	// Only enabled zones are considered
	ELSIF ZoneTable[mIdx].Used THEN
		// Only empty zones are considered and not marked to be flushed
		IF NOT ZoneTable[mIdx].TU_Present AND NOT ZoneTable[mIdx].Flush THEN
			// A zone candidate needs to provide the right length and is not reserver already
			IF ZoneTable[mIdx].ActionId = 0 AND
               ZoneTable[mIdx].ZoneLength >=  mLength THEN
				// When start position of zone is higher, the position is in front of the requested position
				// All others are after overflow point
				IF ZoneTable[mIdx].ZoneStartPosition >= mTrackingPosition THEN
					mDistanceToCurrentZone := ZoneTable[mIdx].ZoneStartPosition - mTrackingPosition;
					
					// Check if distance in a valid range for assignment
					IF mDistanceToCurrentZone <= mMaxAssignDistance THEN
						IF mDistanceToLastFoundZone > mDistanceToCurrentZone THEN
							mDistanceToLastFoundZone := mDistanceToCurrentZone;
							mFoundZoneIndex := mIdx;
						END_IF
					END_IF
				ELSE
					mDistanceToCurrentZone := ZoneTable[mIdx].ZoneStartPosition + TotalTrackingLength - mTrackingPosition;
				
					// Check if distance in a valid range for assignment
					IF mDistanceToCurrentZone <= mMaxAssignDistance THEN
						IF mDistanceToLastFoundZone > mDistanceToCurrentZone THEN
							mDistanceToLastFoundZone := mDistanceToCurrentZone;
							mFoundZoneIndex := mIdx;
						END_IF
					END_IF
				END_IF
			END_IF
		END_IF
		
		mZoneCounter := mZoneCounter + 1;
	END_IF	
END_FOR

// Reserve zone
IF mFoundZoneIndex > 0 THEN
	ZoneTable[mFoundZoneIndex].ActionId := mActionId;
	ZoneTable[mFoundZoneIndex].iActionListener := miActionListener;
	ZoneTable[mFoundZoneIndex].PositionToLive := mPositionToLive;
	
	// When a position to live is configured, ensure zone gets monitored
	IF mPositionToLive > 0 THEN
		M_AddZoneToPTL(mFoundZoneIndex);
	ELSE
		// It is possible that found zone had already a PTL
		// If new one is 0, means no monitoring
		M_RemoveZoneFromPTL(mFoundZoneIndex);
	END_IF
END_IF

M_AssignNextFreeZone := mFoundZoneIndex;
END_METHOD

/// Calculates full tracking distance and ensure its a multiple of windowsize.
/// Additional it adds the tracking addition distance to allow more space for reservations.
METHOD PROTECTED M_CalculateTotalTrackingLength : UDINT // Returns complete tracking distance 
VAR_INPUT
	mTrackingLength			: UDINT; // Length of tracking segment [mm] (e.g. conveyor length)
	mTrackingAddition		: UDINT; // Additional tracking length [mm]
	mWindowSize				: UINT; // Window size [mm]
END_VAR
VAR
	mLength					: UDINT; // Tracking length with out taking care of window size
	mRest					: UDINT; // Missing value between Length and next integer
END_VAR
(* Calculation is based on the following:
	+ 2 * Tracking length
	+ Tracking addition
	+ supplement to ensure its a multiple of window size
*)

mLength := mTrackingLength * 2 + TrackingAddition;
mRest := mLength MOD mWindowSize;

IF mRest > 0 THEN
	M_CalculateTotalTrackingLength := mLength + (mWindowSize-mRest);
ELSE
	M_CalculateTotalTrackingLength := mLength;
END_IF
END_METHOD

/// Clears all windows, zones and ongoing transfers. Notifies all listeners.
/// Remark: This method is executed immediately and can therefore influence
///         ongoing operations.
METHOD M_ClearTables : BOOL // Returns true if successful, otherwise false
VAR
	mZoneCounter		: INT;
	mIdx				: UINT;
END_VAR
VAR_INST
	AllTablesCleared	: BOOL;
	OldZoneTable		: ARRAY[1..MAX_NUMBER_OF_ZONES] OF ST_WindowTrackingZone; // List of all zones
END_VAR
M_ClearTables := FALSE;

// Store old zone table
OldZoneTable := ZoneTable;

// Clear all tables
AllTablesCleared := MEMSET(ADR(WindowTable), 0, SIZEOF(WindowTable)) > 0 AND
				    MEMSET(ADR(ZoneTable), 0, SIZEOF(ZoneTable)) > 0 AND
				    MEMSET(ADR(OngoingTransferList), 0, SIZEOF(OngoingTransferList)) > 0 AND
				    MEMSET(ADR(PTL_Zones), 0, SIZEOF(PTL_Zones)) > 0;

// Inform listener
IF AllTablesCleared THEN
	mZoneCounter := 0;
	// Notify listeners
	FOR mIdx := 1 TO MAX_NUMBER_OF_ZONES DO
		// When number of present zone is reached
		IF mZoneCounter >= ZoneCount THEN
			EXIT;
			
		ELSIF OldZoneTable[mIdx].Used THEN
			// Check if zone had a registred action lister and notify
			IF OldZoneTable[mIdx].iActionListener <> 0 THEN
				OldZoneTable[mIdx].iActionListener.M_ActionZoneDeletedEvent(mIdx,OldZoneTable[mIdx]);
			END_IF
			
			// Inform window tracking listener
			IF iEventListener <> 0 THEN
				IF OldZoneTable[mIdx].TU_Present THEN
					iEventListener.M_TrackingTU_DeletedEvent(mIdx,OldZoneTable[mIdx]);
				END_IF
				
				iEventListener.M_TrackingZoneDeletedEvent(mIdx,OldZoneTable[mIdx]);
			END_IF
	
			mZoneCounter := mZoneCounter + 1;	
		END_IF
	END_FOR
	
	// Clean internal counters
	ZoneCount := 0;
	TU_Count := 0;
	
	M_ClearTables := TRUE;
END_IF
END_METHOD

/// Clears window and initialize with default values
METHOD PROTECTED M_ClearWindow : BOOL // returns true if successfull cleared, otherwise false
VAR_INPUT
	mWindowIndex	: UINT; // Window index to clear
END_VAR
M_ClearWindow := FALSE;

// Validate inputs
IF mWindowIndex <= 0 OR
   mWindowIndex > MaxWindowIndex THEN
   RETURN;
END_IF

M_ClearWindow := MEMSET(ADR(WindowTable[mWindowIndex]), 0, SIZEOF(WindowTable[mWindowIndex])) > 0;
END_METHOD

/// Delete a zone and all related windows
/// Remark: Including zones with physical TUs 
METHOD M_DeleteZone : BOOL // Returns true if successful, otherwise false
VAR_INPUT
	mZoneIndex 				: UINT; // Zone index to delete
END_VAR
VAR
	mIdx					: UINT; // Loop iterator
	mZoneWindowLength 		: UINT; // Length of zone to be moved
	mWindowIndex			: UINT; // Start window index
	mDeletedOnTransferList	: BOOL; // Zone was found and deleted on transfer list
	mDeletedOnPTL			: BOOL; // Zone was found and deleted in PTL list
END_VAR
VAR_INST
	OldZoneData				: ST_WindowTrackingZone; // Old deleted zone data
END_VAR
M_DeleteZone := FALSE;

// Validate inputs
IF mZoneIndex <= 0 OR
   mZoneIndex > MAX_NUMBER_OF_ZONES THEN
   RETURN;
END_IF

// Check if zone is complete
IF ZoneTable[mZoneIndex].ZoneEndWindowIndex > 0 AND
   ZoneTable[mZoneIndex].ZoneStartWindowIndex > 0 THEN
	
	// Calculate length of zone to move
	IF ZoneTable[mZoneIndex].ZoneEndWindowIndex >= ZoneTable[mZoneIndex].ZoneStartWindowIndex THEN
		mZoneWindowLength := ZoneTable[mZoneIndex].ZoneEndWindowIndex - ZoneTable[mZoneIndex].ZoneStartWindowIndex + 1;
	ELSE
		mZoneWindowLength := ZoneTable[mZoneIndex].ZoneEndWindowIndex + MaxWindowIndex - ZoneTable[mZoneIndex].ZoneStartWindowIndex + 1;
	END_IF
		
// Otherwise scan all windows
ELSE
	mZoneWindowLength := MaxWindowIndex;
END_IF

// When start is known, start deleting of windows
IF ZoneTable[mZoneIndex].ZoneStartWindowIndex > 0 THEN
	mWindowIndex := ZoneTable[mZoneIndex].ZoneStartWindowIndex;
	// Store zone data for report
	OldZoneData := ZoneTable[mZoneIndex];
	
	// Loop through all windows and delete them
	FOR mIdx := 1 TO mZoneWindowLength DO
		// Ensure that window is part of requested zone
		IF WindowTable[mWindowIndex].ZoneIndex = mZoneIndex THEN
			// Delete window
			M_ClearWindow(mWindowIndex);
		// Otherwise stop deleting
		ELSE
			EXIT;
		END_IF
		
		mWindowIndex := mWindowIndex + 1;
		 
		// Correct border overflow
		IF mWindowIndex > MaxWindowIndex THEN
			mWindowIndex := mWindowIndex - MaxWindowIndex;
		END_IF
	END_FOR
END_IF

// When zone had a TU present, update counter values
IF ZoneTable[mZoneIndex].TU_Present THEN
	TU_Count := TU_Count - 1;
	
	IF TU_Count < 0 THEN
		TU_Count := 0;
	END_IF
	
	// Inform listener
	IF iEventListener <> 0 THEN
		iEventListener.M_TrackingTU_DeletedEvent(mZoneIndex,OldZoneData);
	END_IF
END_IF

// Clean entry in transfer list and close gaps in list
mDeletedOnTransferList := M_RemoveZoneFromTransferList(mZoneIndex);
mDeletedOnPTL := M_RemoveZoneFromPTL(mZoneIndex);

// Delete Zone Index
MEMSET(ADR(ZoneTable[mZoneIndex]),0,SIZEOF(ZoneTable[mZoneIndex]));

ZoneCount := ZoneCount - 1;

IF ZoneCount < 0 THEN
	ZoneCount := 0;
END_IF

// Inform listener
IF iEventListener <> 0 THEN
	iEventListener.M_TrackingZoneDeletedEvent(mZoneIndex,OldZoneData);
END_IF

// Check if zone had a registred action listener and notify
IF OldZoneData.iActionListener <> 0 THEN
	OldZoneData.iActionListener.M_ActionZoneDeletedEvent(mZoneIndex,OldZoneData);
END_IF

// If the currently monitored index is same as the deleted one, reset monitoring
IF EndZoneIndex = mZoneIndex THEN
	EndZoneIndex := 0;
END_IF

M_DeleteZone := TRUE;
END_METHOD

/// Enlarges a zone by given value in up- or downstream direction
METHOD M_EnlargeZone : BOOL// Returns TRUE if successful,
VAR_INPUT
	mZoneIndex 				: UINT; // Zone index to enlarge
	mAdditionalLength		: UINT; // Add this length to existing zone [mm]
	mShiftFrontEdge			: BOOL; // Shift front edge for enlargement
END_VAR
VAR
	mIdx					: UINT; // Loop iterator
	mWindowIndex			: UINT; // Start window index
	mAdditionalWindowLength	: UINT; // Zone length in windows
	mEnlargementAllowed 	: BOOL; // Enlargement valid (e.g. free space available)
	mZoneEndWindowIndex		: UINT; // Zone end window index
	mZoneStartWindowIndex	: UINT; // Zone start window index
	mFreeOK					: BOOL; // Free operation successful
	mZoneEndPositionNew		: UDINT; // Zone end position after enlargement
	mZoneStartPositionNew	: UDINT; // Zone start position after enlargement
END_VAR
VAR_INST
	OldZoneData				: ST_WindowTrackingZone; // Old tracking zone data
END_VAR
M_EnlargeZone := FALSE;

// Validate inputs
IF mZoneIndex <= 0 OR
   mZoneIndex > MAX_NUMBER_OF_ZONES OR
   WindowSize = 0 THEN
   RETURN;
END_IF

IF NOT mShiftFrontEdge THEN
	// Calculate new zone end position
	IF ZoneTable[mZoneIndex].ZoneEndPosition + mAdditionalLength > TotalTrackingLength THEN
		mZoneEndPositionNew := ZoneTable[mZoneIndex].ZoneEndPosition + mAdditionalLength - TotalTrackingLength;
		mAdditionalWindowLength := M_GetWindowIndex(M_GetAbsolutePosition(mZoneEndPositionNew)) - M_GetWindowIndex(M_GetAbsolutePosition(ZoneTable[mZoneIndex].ZoneEndPosition)) + MaxWindowIndex;
	ELSE
		mZoneEndPositionNew := ZoneTable[mZoneIndex].ZoneEndPosition + mAdditionalLength;
		mAdditionalWindowLength := M_GetWindowIndex(M_GetAbsolutePosition(mZoneEndPositionNew)) - M_GetWindowIndex(M_GetAbsolutePosition(ZoneTable[mZoneIndex].ZoneEndPosition));
	END_IF

	mWindowIndex := ZoneTable[mZoneIndex].ZoneEndWindowIndex;
	mEnlargementAllowed := TRUE;
	
	// Ensure reservation is possible
	FOR mIdx := 1 TO mAdditionalWindowLength DO
		mWindowIndex := mWindowIndex + 1;
	 
		// Correct border overflow
		IF mWindowIndex > MaxWindowIndex THEN
			mWindowIndex := mWindowIndex - MaxWindowIndex;
		END_IF
		
		// Is on intended window index already part of a zone, try to shift
		IF WindowTable[mWindowIndex].ZoneIndex > 0 THEN
			// Shift reserved zones
			mFreeOK := M_MakeSpace(mWindowIndex, 1, FALSE);
			
			IF NOT mFreeOK THEN
			   // Cancel reservation
			   mEnlargementAllowed := FALSE;
			   M_EnlargeZone := FALSE;
		   
				// Error
				fbDebugMsg.M_SendErrorMsg('M_EnlargeZone - Enlargement not possible, no available space.');	
				RETURN;
			END_IF
		END_IF	
	END_FOR
ELSE
	// Calculate new zone start position
	IF mAdditionalLength > ZoneTable[mZoneIndex].ZoneStartPosition THEN
		mZoneStartPositionNew := ZoneTable[mZoneIndex].ZoneStartPosition - mAdditionalLength + TotalTrackingLength;
		mAdditionalWindowLength := M_GetWindowIndex(M_GetAbsolutePosition(ZoneTable[mZoneIndex].ZoneStartPosition)) - M_GetWindowIndex(M_GetAbsolutePosition(mZoneStartPositionNew)) + MaxWindowIndex;
	ELSE
		mZoneStartPositionNew := ZoneTable[mZoneIndex].ZoneStartPosition + mAdditionalLength;
		mAdditionalWindowLength := M_GetWindowIndex(M_GetAbsolutePosition(ZoneTable[mZoneIndex].ZoneStartPosition)) - M_GetWindowIndex(M_GetAbsolutePosition(mZoneStartPositionNew));
	END_IF
	
	mWindowIndex := ZoneTable[mZoneIndex].ZoneStartWindowIndex;
	mEnlargementAllowed := TRUE;
	
	// Ensure reservation is possible
	FOR mIdx := 1 TO mAdditionalWindowLength DO
		mWindowIndex := mWindowIndex - 1;
	 
		// Correct border overflow
		IF mWindowIndex = 0 THEN
			mWindowIndex := MaxWindowIndex;
		END_IF
		
		// Is on intended window index already part of a zone, try to shift
		IF WindowTable[mWindowIndex].ZoneIndex > 0 THEN
			// Cancel reservation
			mEnlargementAllowed := FALSE;
			M_EnlargeZone := FALSE;
		   
			// Error
			fbDebugMsg.M_SendErrorMsg('M_EnlargeZone - Enlargement not possible, no available space.');	
			RETURN;
		END_IF	
	END_FOR
END_IF

// When enlargement is possible to be executed
IF mEnlargementAllowed THEN
	
	OldZoneData := ZoneTable[mZoneIndex];

	IF NOT mShiftFrontEdge THEN
		mWindowIndex := ZoneTable[mZoneIndex].ZoneEndWindowIndex;
		// Init
		mZoneEndWindowIndex := mWindowIndex;
		
		// Loop through all windows and assign new zone
		FOR mIdx := 1 TO mAdditionalWindowLength DO
			mWindowIndex := mWindowIndex + 1;
		 
			// Correct border overflow
			IF mWindowIndex > MaxWindowIndex THEN
				mWindowIndex := mWindowIndex - MaxWindowIndex;
			END_IF
			
		   // Clear window
			MEMSET(ADR(WindowTable[mWindowIndex]), 0, SIZEOF(WindowTable[mWindowIndex]));
			
			WindowTable[mWindowIndex].ZoneIndex := mZoneIndex;
			WindowTable[mWindowIndex].State := E_WindowTrackingWindowState.RESERVED;
							
			mZoneEndWindowIndex := mWindowIndex;
		END_FOR	
		
		// Update zone table
		ZoneTable[mZoneIndex].ZoneEndWindowIndex := mZoneEndWindowIndex;
		ZoneTable[mZoneIndex].ZoneEndPosition := mZoneEndPositionNew;
		ZoneTable[mZoneIndex].ZoneLength := ZoneTable[mZoneIndex].ZoneLength + mAdditionalLength;
		
		// Inform listener
		IF iEventListener <> 0 THEN
			iEventListener.M_TrackingZoneEnlargedEvent(
				mTrackingZoneIndex 		:= mZoneIndex,
                mOldTrackingZoneData 	:= OldZoneData,
                mNewTrackingZoneDAta 	:= ZoneTable[mZoneIndex]);
		END_IF
		
		M_EnlargeZone := TRUE;
	ELSE
		mWindowIndex := ZoneTable[mZoneIndex].ZoneStartWindowIndex;
			
		// Loop through all windows and assign new zone
		// Init
		mZoneStartWindowIndex := mWindowIndex;
		
		FOR mIdx := 1 TO mAdditionalWindowLength DO
			mWindowIndex := mWindowIndex - 1;
		 
			// Correct border overflow
			IF mWindowIndex = 0 THEN
				mWindowIndex := MaxWindowIndex;
			END_IF
			
		   // Clear window
			MEMSET(ADR(WindowTable[mWindowIndex]), 0, SIZEOF(WindowTable[mWindowIndex]));
			
			WindowTable[mWindowIndex].ZoneIndex := mZoneIndex;
			WindowTable[mWindowIndex].State := E_WindowTrackingWindowState.RESERVED;
							
			mZoneStartWindowIndex := mWindowIndex;
		END_FOR		
		
		// Update zone table
		ZoneTable[mZoneIndex].ZoneStartWindowIndex := mZoneStartWindowIndex;
		ZoneTable[mZoneIndex].ZoneStartPosition := mZoneStartPositionNew;
		ZoneTable[mZoneIndex].ZoneLength := ZoneTable[mZoneIndex].ZoneLength + mAdditionalLength;
		
		// Inform listener
		IF iEventListener <> 0 THEN
			iEventListener.M_TrackingZoneEnlargedEvent(
				mTrackingZoneIndex 		:= mZoneIndex,
                mOldTrackingZoneData 	:= OldZoneData,
                mNewTrackingZoneDAta 	:= ZoneTable[mZoneIndex]);
		END_IF
		
		M_EnlargeZone := TRUE;
	END_IF
END_IF
END_METHOD

/// Marks all windows and zones in an area to be flushed.
/// (e.g. because of an error the TU position is not reliable anymore)
/// Remark: This includes empty windows as well
METHOD M_FlushDistance : BOOL // Returns true if successful, otherwise false
VAR_INPUT
	mAbsoluteStartPosition		: UDINT; // Position to start marking [mm]
	mAbsoluteEndPosition		: UDINT; // Position to stop marking [mm]
END_VAR
VAR
	mStartWindowIndex			: UINT; // Start window index
	mEndWindowIndex				: UINT; // End window index
	mWindowLength				: UINT; // Window length
	mWindowIndex				: UINT; // Window index iterator
	mZoneIndex					: UINT; // Zone index of window
	mIdx						: UINT; // Loop iterator
END_VAR
M_FlushDistance := FALSE;

mEndWindowIndex := M_GetWindowIndex(mAbsoluteStartPosition);
mStartWindowIndex := M_GetWindowIndex(mAbsoluteEndPosition);

IF mEndWindowIndex > mStartWindowIndex THEN
	mWindowLength := mEndWindowIndex - mStartWindowIndex + 1;
ELSE
	mWindowLength := mEndWindowIndex + MaxWindowIndex - mStartWindowIndex + 1;
END_IF

mWindowIndex := mStartWindowIndex;

FOR mIdx := 1 TO mWindowLength DO
	WindowTable[mWindowIndex].Flush := TRUE;
	
	// If window is part of zone, mark full zone as to be flushed
	IF WindowTable[mWindowIndex].ZoneIndex > 0 THEN
		mZoneIndex := WindowTable[mWindowIndex].ZoneIndex;
		
		ZoneTable[mZoneIndex].Flush := TRUE;
	END_IF

	mWindowIndex := mWindowIndex + 1;
	
	// Correct window border overflow
	IF mWindowIndex > MaxWindowIndex THEN
		mWindowIndex := mWindowIndex - MaxWindowIndex;
	END_IF
END_FOR

M_FlushDistance := TRUE;
END_METHOD

/// Converts a tracking position into the absolute position regarding tracking length
METHOD M_GetAbsolutePosition : UDINT // Absolute position releated to Tracking length [mm]
VAR_INPUT
	mTrackingPosition			: UDINT; // Tracking position on tracking 
END_VAR
VAR
	mCurrentEncoderPosition		: UDINT; // Current tracking position [mm]
	mRequestingTrackingPosition : UDINT; // Requesting position on tracking [mm]
END_VAR
mCurrentEncoderPosition := (TrackingPosition MOD TotalTrackingLength);
mRequestingTrackingPosition := (mTrackingPosition MOD TotalTrackingLength);

IF mRequestingTrackingPosition < mCurrentEncoderPosition THEN
	M_GetAbsolutePosition := mCurrentEncoderPosition - mRequestingTrackingPosition;
ELSE
	M_GetAbsolutePosition := mCurrentEncoderPosition - mRequestingTrackingPosition + TotalTrackingLength;
END_IF
END_METHOD

/// Returns distance to end of tu from observation point. 
/// Position 0 = observation point, Position Max = Observation point plus half tracking length.
/// Remark: In order to reduce the area use M_IsZoneInRange.
METHOD M_GetDistanceToTU_End : DINT // Returns distance to tu end. x < 0 Zone has already passed by x
VAR_INPUT
	mAbsolutePosition		: UDINT; // Absolute position to watch
	mZoneIndex				: UINT; // Index to be measured
END_VAR
VAR
	mTrackingPosition		: DINT; // Current position on tracking
	mTU_EndPosition			: DINT; // TU end tracking position
	mEndWindowIndex			: UINT; // End window index
	mDistanceAhead			: DINT; // Distance to zone ahead
	mDistanceAfter			: DINT; // Distance to zone after
END_VAR
M_GetDistanceToTU_End := 0;

// Validate inputs
IF mZoneIndex <= 0 OR
   mZoneIndex > MAX_NUMBER_OF_ZONES THEN
	RETURN;
END_IF

IF NOT ZoneTable[mZoneIndex].Used OR
  ZoneTable[mZoneIndex].TU_EndWindowIndex = 0 THEN
	RETURN;
END_IF

// Get position of observation point on tracking (=0)
mTrackingPosition := UDINT_TO_DINT(M_GetTrackingPosition(mAbsolutePosition));
mEndWindowIndex := ZoneTable[mZoneIndex].TU_EndWindowIndex;

mTU_EndPosition := UDINT_TO_DINT(WindowTable[mEndWindowIndex].TU_RearEdgePosition);

// Calculate distance in both directions, Zone is ahead to observation point or after
mDistanceAhead := (mTU_EndPosition - mTrackingPosition + UDINT_TO_DINT(TotalTrackingLength)) MOD UDINT_TO_DINT(TotalTrackingLength);
mDistanceAfter := (mTrackingPosition - mTU_EndPosition + UDINT_TO_DINT(TotalTrackingLength)) MOD UDINT_TO_DINT(TotalTrackingLength);

// Definition range: Ahead = + / After = -
// Ahead = Max -1 -> Observation
// After = Observation -> Max
IF mDistanceAfter <= mDistanceAhead THEN
	M_GetDistanceToTU_End := mDistanceAfter * (-1);
ELSE
	M_GetDistanceToTU_End := mDistanceAhead;
END_IF
END_METHOD

/// Returns distance to begin of TU from observation point. 
/// Position 0 = observation point, Position Max = Observation point plus half tracking length.
/// Remark: In order to reduce the area use M_IsZoneInRange.
METHOD M_GetDistanceToTU_Start : DINT // Returns distance to tu start. x < 0 Zone has already passed by x
VAR_INPUT
	mAbsolutePosition		: UDINT; // Absolute position to watch
	mZoneIndex				: UINT; // Index to be measured
END_VAR
VAR
	mTrackingPosition		: DINT; // Current position on tracking
	mTU_StartPosition		: DINT; // TU start tracking position
	mStartWindowIndex		: UINT; // Start window index
	mDistanceAhead			: DINT; // Distance to zone ahead
	mDistanceAfter			: DINT; // Distance to zone after
END_VAR
M_GetDistanceToTU_Start := 0;

// Validate inputs
IF mZoneIndex <= 0 OR
   mZoneIndex > MAX_NUMBER_OF_ZONES THEN
	RETURN;
END_IF

IF NOT ZoneTable[mZoneIndex].Used OR
  ZoneTable[mZoneIndex].TU_StartWindowIndex = 0 THEN
	RETURN;
END_IF

// Get position of observation point on tracking (=0)
mTrackingPosition := UDINT_TO_DINT(M_GetTrackingPosition(mAbsolutePosition));
mStartWindowIndex := ZoneTable[mZoneIndex].TU_StartWindowIndex;

mTU_StartPosition := UDINT_TO_DINT(WindowTable[mStartWindowIndex].TU_FrontEdgePosition);

// Calculate distance in both directions, Zone is ahead to observation point or after
mDistanceAhead := (mTU_StartPosition - mTrackingPosition + UDINT_TO_DINT(TotalTrackingLength)) MOD UDINT_TO_DINT(TotalTrackingLength);
mDistanceAfter := (mTrackingPosition - mTU_StartPosition + UDINT_TO_DINT(TotalTrackingLength)) MOD UDINT_TO_DINT(TotalTrackingLength);

// Definition range: Ahead = + / After = -
// Ahead = Max -1 -> Observation
// After = Observation -> Max
IF mDistanceAfter <= mDistanceAhead THEN
	M_GetDistanceToTU_Start := mDistanceAfter * (-1);
ELSE
	M_GetDistanceToTU_Start := mDistanceAhead;
END_IF
END_METHOD

/// Returns distance to end of zone from observation point. 
/// Position 0 = observation point, Position Max = Observation point plus half tracking length.
/// Remark: In order to reduce the area use M_IsZoneInRange.
METHOD M_GetDistanceToZoneEnd : DINT // Returns distance to zone end. x < 0 Zone has already passed by x
VAR_INPUT
	mAbsolutePosition		: UDINT; // Absolute position to watch
	mZoneIndex				: UINT; // Index to be measured
END_VAR
VAR
	mTrackingPosition		: DINT; // Current position on tracking
	mZoneEndPosition		: DINT; // Zone end tracking position
	mDistanceAhead			: DINT; // Distance to zone ahead
	mDistanceAfter			: DINT; // Distance to zone after
END_VAR
M_GetDistanceToZoneEnd := 0;

// Validate inputs
IF mZoneIndex <= 0 OR
   mZoneIndex > MAX_NUMBER_OF_ZONES THEN
	RETURN;
END_IF

IF NOT ZoneTable[mZoneIndex].Used THEN
	RETURN;
END_IF

// Get position of observation point on tracking (=0)
mTrackingPosition := UDINT_TO_DINT(M_GetTrackingPosition(mAbsolutePosition));
mZoneEndPosition := UDINT_TO_DINT(ZoneTable[mZoneIndex].ZoneEndPosition);

// Calculate distance in both directions, Zone is ahead to observation point or after
mDistanceAhead := (mZoneEndPosition - mTrackingPosition + UDINT_TO_DINT(TotalTrackingLength)) MOD UDINT_TO_DINT(TotalTrackingLength);
mDistanceAfter := (mTrackingPosition - mZoneEndPosition + UDINT_TO_DINT(TotalTrackingLength)) MOD UDINT_TO_DINT(TotalTrackingLength);

// Definition range: Ahead = + / After = -
// Ahead = Max -1 -> Observation
// After = Observation -> Max
IF mDistanceAfter <= mDistanceAhead THEN
	M_GetDistanceToZoneEnd := mDistanceAfter * (-1);
ELSE
	M_GetDistanceToZoneEnd := mDistanceAhead;
END_IF
END_METHOD

/// Returns distance to begin of zone from observation point. 
/// Position 0 = observation point, Position Max = Observation point plus half tracking length.
/// Remark: In order to reduce the area use M_IsZoneInRange.
METHOD M_GetDistanceToZoneStart : DINT // Returns distance [mm] to zone start. x < 0 Zone has already passed by x
VAR_INPUT
	mAbsolutePosition		: UDINT; // Absolute position to watch
	mZoneIndex				: UINT; // Index to be measured
END_VAR
VAR
	mTrackingPosition		: DINT; // Current position on tracking
	mZoneStartPosition		: DINT; // Zone start tracking position
	mDistanceAhead			: DINT; // Distance to zone ahead
	mDistanceAfter			: DINT; // Distance to zone after
END_VAR
M_GetDistanceToZoneStart := 0;

// Validate inputs
IF mZoneIndex <= 0 OR
   mZoneIndex > MAX_NUMBER_OF_ZONES THEN
	RETURN;
END_IF

IF NOT ZoneTable[mZoneIndex].Used THEN
	RETURN;
END_IF

// Get position of observation point on tracking (=0)
mTrackingPosition := UDINT_TO_DINT(M_GetTrackingPosition(mAbsolutePosition));
mZoneStartPosition := UDINT_TO_DINT(ZoneTable[mZoneIndex].ZoneStartPosition);

// Calculate distance in both directions, Zone is ahead to observation point or after
mDistanceAhead := (mZoneStartPosition - mTrackingPosition + UDINT_TO_DINT(TotalTrackingLength)) MOD UDINT_TO_DINT(TotalTrackingLength);
mDistanceAfter := (mTrackingPosition - mZoneStartPosition + UDINT_TO_DINT(TotalTrackingLength)) MOD UDINT_TO_DINT(TotalTrackingLength);

// Definition range: Ahead = + / After = -
// Ahead = Max -1 -> Observation
// After = Observation -> Max
IF mDistanceAfter <= mDistanceAhead THEN
	M_GetDistanceToZoneStart := mDistanceAfter * (-1);
ELSE
	M_GetDistanceToZoneStart := mDistanceAhead;
END_IF
END_METHOD

/// Returns first zone index that can be found between start and end position, direction according windows ascending
/// REMARK: Size of area to be checked has influence to performance of method
METHOD M_GetFirstZoneIndex : UINT // Returns ZoneIndex > 0, otherwise 0
VAR_INPUT
	mAbsoluteStartPosition	: UDINT; // Start position on the tracking [mm]
	mAbsoluteEndPosition	: UDINT; // End position on the tracking [mm]
	mOnlyZonesWithTU		: BOOL; // Check only zones with physical TU
END_VAR
VAR
	mIdx					: UINT; // Iterator
	mStartWindowIndex		: UINT; // Window index at start position
	mEndWindowIndex			: UINT; // Window index at end position
	mWindowLength 			: UINT; // Length of are to be checked in windows
	mWindowIndex 			: UINT; // Window interator
	mTrackingPositionEnd	: UDINT; // Tracking position end
	mTrackingPositionStart	: UDINT; // Tracking position start
	mZoneIndex				: UINT; // Tracking zone index
END_VAR
M_GetFirstZoneIndex := 0;

// Get window index of window start position
mStartWindowIndex := M_GetWindowIndex(mAbsoluteStartPosition);
// Get window index of window end position
mEndWindowIndex := M_GetWindowIndex(mAbsoluteEndPosition);

// Remark:
// Absolute view is unequal to tracking view
// ABS:  500mm 505mm .....1000mm
//    Startpos			 EndPos
//       |                  |
//  --------------------------------------      FlowDirection ->
// Win:  54  53  52 ....  43 42 ...
// Window index of end is normally lower than start (except overflow)     

// Ensure both window index are in a valid range
IF mStartWindowIndex > 0 AND mStartWindowIndex <= WindowTracking.MAX_NUMBER_OF_WINDOWS AND
   mEndWindowIndex > 0 AND mEndWindowIndex <= WindowTracking.MAX_NUMBER_OF_WINDOWS THEN
	
   	mTrackingPositionStart := M_GetTrackingPosition(mAbsoluteStartPosition);
   	mTrackingPositionEnd := M_GetTrackingPosition(mAbsoluteEndPosition);
   
	// Calculate windows to check
	IF mStartWindowIndex >= mEndWindowIndex THEN
		mWindowLength := mStartWindowIndex - mEndWindowIndex + 1;
	ELSE
		mWindowLength := mStartWindowIndex + MaxWindowIndex - mEndWindowIndex + 1;
	END_IF
	
	mWindowIndex := mStartWindowIndex;

	FOR mIdx := 1 TO mWindowLength DO
		mZoneIndex := WindowTable[mWindowIndex].ZoneIndex;
		// Search for zone
		IF mZoneIndex > 0 THEN
			// If search is limited to physically occupied zone
			IF mOnlyZonesWithTU THEN
				// When the currently checked window is the start window (EndWindowIndex) of the checked
				// range and at the same time the rear edge of a TU, check exact position
				// in window
				IF mWindowIndex = mEndWindowIndex AND
				   WindowTable[mWindowIndex].State = E_WindowTrackingWindowState.REAR_EDGE THEN
				   // Check exact position of zone end
				   IF WindowTable[mWindowIndex].TU_RearEdgePosition >= mTrackingPositionEnd THEN
					   M_GetFirstZoneIndex := WindowTable[mWindowIndex].ZoneIndex;
					   RETURN;
				   END_IF
				   
				// When the currently checked window is the end window (StartWindowIndex) of the checked
				// range and at the same time the front edge of a TU, check exact position
				// in window
				ELSIF mWindowIndex = mStartWindowIndex AND
					  WindowTable[mWindowIndex].State = E_WindowTrackingWindowState.FRONT_EDGE THEN
					// Check exact position of zone end
				   IF WindowTable[mWindowIndex].TU_FrontEdgePosition <= mTrackingPositionStart THEN
					   M_GetFirstZoneIndex := WindowTable[mWindowIndex].ZoneIndex;
					   RETURN;
				   END_IF
				   
				// When window is occupied, its completly part of the TU
				ELSIF WindowTable[mWindowIndex].State = E_WindowTrackingWindowState.OCCUPIED THEN
					// Check begin of zone
					M_GetFirstZoneIndex := WindowTable[mWindowIndex].ZoneIndex;
					RETURN;
				END_IF
			ELSE
				// When the currently checked window is the start window (EndWindowIndex) of the checked
				// range and at the same time the end window of a zone, check exact position
				// in window
				IF mWindowIndex = mEndWindowIndex AND
				   mWindowIndex = ZoneTable[mZoneIndex].ZoneEndWindowIndex THEN
				   // Check exact position of zone end
				   IF ZoneTable[mZoneIndex].ZoneEndPosition >= mTrackingPositionEnd THEN
					   M_GetFirstZoneIndex := WindowTable[mWindowIndex].ZoneIndex;
					   RETURN;
				   END_IF
				   
				// When the currently checked window is the end window (StartWindowIndex) of the checked
				// range and at the same time the start window of a zone, check exact position
				// in window
				ELSIF mWindowIndex = mStartWindowIndex AND
					  mWindowIndex = ZoneTable[mZoneIndex].ZoneStartWindowIndex THEN
					// Check exact position of zone end
				   IF ZoneTable[mZoneIndex].ZoneStartPosition <= mTrackingPositionStart THEN
					   M_GetFirstZoneIndex := WindowTable[mWindowIndex].ZoneIndex;
					   RETURN;
				   END_IF
				   
				// Otherwise the zone uses the whole window
				ELSE
					M_GetFirstZoneIndex := WindowTable[mWindowIndex].ZoneIndex;
					RETURN;
				END_IF
			END_IF
		END_IF	
		
		mWindowIndex := mWindowIndex - 1;
			
		// Correct border overflow
		IF mWindowIndex <= 0 THEN
			mWindowIndex := mWindowIndex + MaxWindowIndex;
		END_IF
	END_FOR
END_IF
END_METHOD

/// Returns last zone index that can be found between start and end position, direction according windows ascending
/// REMARK: Size of area to be checked has influence to performance of method
METHOD M_GetLastZoneIndex : UINT // Returns ZoneIndex > 0, otherwise 0
VAR_INPUT
	mAbsoluteStartPosition	: UDINT; // Start position on the tracking [mm]
	mAbsoluteEndPosition	: UDINT; // End position on the tracking [mm]
	mOnlyZonesWithTU		: BOOL; // Check only zones with physical TU in range
END_VAR
VAR
	mIdx					: UINT; // Iterator
	mStartWindowIndex		: UINT; // Window index at start position
	mEndWindowIndex			: UINT; // Window index at end position
	mWindowLength 			: UINT; // Length of are to be checked in windows
	mWindowIndex 			: UINT; // Window interator
	mTrackingPositionEnd	: UDINT; // Tracking position end
	mTrackingPositionStart	: UDINT; // Tracking position start
	mZoneIndex				: UINT; // Tracking zone index
END_VAR
M_GetLastZoneIndex := 0;

// Get window index of window start position
mStartWindowIndex := M_GetWindowIndex(mAbsoluteStartPosition);
// Get window index of window end position
mEndWindowIndex := M_GetWindowIndex(mAbsoluteEndPosition);

// Remark:
// Absolute view is unequal to tracking view
// ABS:  500mm 505mm .....1000mm
//    Startpos			 EndPos
//       |                  |
//  --------------------------------------      FlowDirection ->
// Win:  54  53  52 ....  43 42 ...
// Window index of end is normally lower than start (except overflow)     

// Ensure both window index are in a valid range
IF mStartWindowIndex > 0 AND mStartWindowIndex <= WindowTracking.MAX_NUMBER_OF_WINDOWS AND
   mEndWindowIndex > 0 AND mEndWindowIndex <= WindowTracking.MAX_NUMBER_OF_WINDOWS THEN
	
	mTrackingPositionStart := M_GetTrackingPosition(mAbsoluteStartPosition);
   	mTrackingPositionEnd := M_GetTrackingPosition(mAbsoluteEndPosition);
   
	// Calculate windows to check
	IF mStartWindowIndex >= mEndWindowIndex THEN
		mWindowLength := mStartWindowIndex - mEndWindowIndex + 1;
	ELSE
		mWindowLength := mStartWindowIndex + MaxWindowIndex - mEndWindowIndex + 1;
	END_IF
	
	mWindowIndex := mEndWindowIndex;

	FOR mIdx := 1 TO mWindowLength DO
		mZoneIndex := WindowTable[mWindowIndex].ZoneIndex;
		// Search for zone
		IF mZoneIndex > 0 THEN
			// If search is limited to physically occupied zone
			IF mOnlyZonesWithTU THEN
				// When the currently checked window is the start window (EndWindowIndex) of the checked
				// range and at the same time the rear edge of a TU, check exact position
				// in window
				IF mWindowIndex = mEndWindowIndex AND
				   WindowTable[mWindowIndex].State = E_WindowTrackingWindowState.REAR_EDGE THEN
				   // Check exact position of zone end
				   IF WindowTable[mWindowIndex].TU_RearEdgePosition  >= mTrackingPositionEnd THEN
					   M_GetLastZoneIndex := WindowTable[mWindowIndex].ZoneIndex;
					   RETURN;
				   END_IF
				   
				// When the currently checked window is the end window (StartWindowIndex) of the checked
				// range and at the same time the front edge of a TU, check exact position
				// in window
				ELSIF mWindowIndex = mStartWindowIndex AND
					  WindowTable[mWindowIndex].State = E_WindowTrackingWindowState.FRONT_EDGE THEN
					// Check exact position of zone end
				   IF WindowTable[mWindowIndex].TU_FrontEdgePosition  <= mTrackingPositionStart THEN
					   M_GetLastZoneIndex := WindowTable[mWindowIndex].ZoneIndex;
					   RETURN;
				   END_IF
				   
				// When window is occupied, its completly part of the TU
				ELSIF WindowTable[mWindowIndex].State = E_WindowTrackingWindowState.OCCUPIED THEN
					// Check begin of zone
					M_GetLastZoneIndex := WindowTable[mWindowIndex].ZoneIndex;
					RETURN;
				END_IF
			ELSE
				// When the currently checked window is the start window (EndWindowIndex) of the checked
				// range and at the same time the end window of a zone, check exact position
				// in window
				IF mWindowIndex = mEndWindowIndex AND
				   mWindowIndex = ZoneTable[mZoneIndex].ZoneEndWindowIndex THEN
				   // Check exact position of zone end
				   IF ZoneTable[mZoneIndex].ZoneEndPosition >= mTrackingPositionEnd THEN
					   M_GetLastZoneIndex := WindowTable[mWindowIndex].ZoneIndex;
					   RETURN;
				   END_IF
				   
				// When the currently checked window is the end window (StartWindowIndex) of the checked
				// range and at the same time the start window of a zone, check exact position
				// in window
				ELSIF mWindowIndex = mStartWindowIndex AND
					  mWindowIndex = ZoneTable[mZoneIndex].ZoneStartWindowIndex THEN
					// Check exact position of zone end
				   IF ZoneTable[mZoneIndex].ZoneStartPosition <= mTrackingPositionStart THEN
					   M_GetLastZoneIndex := WindowTable[mWindowIndex].ZoneIndex;
					   RETURN;
				   END_IF
				   
				// Otherwise the zone uses the whole window
				ELSE
					M_GetLastZoneIndex := WindowTable[mWindowIndex].ZoneIndex;
					RETURN;
				END_IF
			END_IF
		END_IF	
		
		mWindowIndex := mWindowIndex + 1;
			
		// Correct border overflow
		IF mWindowIndex > MaxWindowIndex THEN
			mWindowIndex := mWindowIndex - MaxWindowIndex;
		END_IF
	END_FOR
END_IF
END_METHOD

/// Searches through all available zones and add all zone index of ActionId to pData
/// Remark: Amount of available zones has influence to performance.
/// Remark: Existing entries in pData get overwritten.
METHOD M_GetPendingAssignments : BOOL // Returns true if all found zones could be added to pData, otherwise false
VAR_INPUT
	mActionId				: INT; // ID of action which requests zone (<>0)
	mpData 					: POINTER TO UINT; // Address of Value or Array to store the result
	mDataLen				: UINT; // Size of data
END_VAR
VAR_OUTPUT
	mCount					: UINT; // Number of entries added to pData
END_VAR
VAR
	mIdx					: UINT; // Loop iterator
	mZoneIndex				: UINT; // Zone index
	mZoneCounter 			: INT; // Amount of already considerd zones
	mPendingAssignments 	: UINT; // Pending assignments for action id
	mMaxEntries				: UINT; // Max possible entries in offered pData
	mStepSize				: UINT; // Step size between two indexes
	mErrorNoFreeData 		: BOOL; // Error, was not able to add found index to pData
END_VAR
M_GetPendingAssignments := 0;
mZoneIndex := 0;
mCount := 0;
mErrorNoFreeData := FALSE;

// Validate inputs
IF mActionId = 0 OR
   mpData = 0 OR
   mDataLen = 0 THEN
	RETURN;
END_IF

// Abort if no zones available at all
IF ZoneCount = 0 THEN
	M_GetPendingAssignments := 0;
	RETURN;
END_IF

// Calculate max amount of entries that can be assigned of pData
mStepSize := SIZEOF(UINT);
mMaxEntries := mDataLen / mStepSize;

// Clear existing entries
MEMSET(mpData, 0, mDataLen);

mZoneCounter := 0;
mPendingAssignments := 0;

// Check all allocated zones for action id
// Remark: As a reason of performance no scan through all windows upstream is initiated.
FOR mIdx := 1 TO WindowTracking.MAX_NUMBER_OF_ZONES DO
	// When all zones are considered, stop,
	IF mZoneCounter >= ZoneCount THEN
		EXIT;
		
	// Only enabled zones are considered
	ELSIF ZoneTable[mIdx].Used THEN
		// Only empty zones are considered 
		IF NOT ZoneTable[mIdx].TU_Present THEN
			// A zone candidate needs to have required action id
			IF ZoneTable[mIdx].ActionId = mActionId THEN
				// Ensure available memory has still space to be allocated
      			IF mPendingAssignments < mMaxEntries THEN
					// Update value and recalculate next position in pData
					mpData^:= mIdx;
					mpData := mpData + mStepSize;
			
					mPendingAssignments := mPendingAssignments + 1;
				ELSE
					mErrorNoFreeData := TRUE;
					EXIT;
				END_IF
			END_IF
		END_IF
		
		mZoneCounter := mZoneCounter + 1;
	END_IF	
END_FOR

mCount := mPendingAssignments;
M_GetPendingAssignments := NOT mErrorNoFreeData;
END_METHOD

/// Converts an absolute position into the current position on the tracking
METHOD M_GetTrackingPosition : UDINT // Converted position on tracking [mm]
VAR_INPUT
	mAbsolutePosition	: UDINT; // Absolute position 
END_VAR
IF TrackingPosition > mAbsolutePosition THEN
	M_GetTrackingPosition := (TrackingPosition - mAbsolutePosition) MOD TotalTrackingLength;
ELSE
	M_GetTrackingPosition := (TrackingPosition + TotalTrackingLength - mAbsolutePosition) MOD TotalTrackingLength;	
END_IF
END_METHOD

/// Returns TU end position of a zone on tracked distance
/// Remark: User needs to make sure zone is valid
/// Remark: When no TU available the return value is 0, but is notfied with output "NoTuAvailable"
METHOD M_GetTU_EndPosition : UDINT // Returns position of TU end [mm]
VAR_INPUT
	mZoneIndex			: UINT; // Index of zone
END_VAR
VAR_OUTPUT
	mNoTU_Available		: BOOL; // No TU Available
END_VAR
VAR
	mEndWindowIndex		: UINT; // Zone end window index
	mPositionOnTracking	: UDINT; // Position on tracking length
END_VAR
M_GetTU_EndPosition := 0;
mNoTU_Available := FALSE;
mEndWindowIndex := 0;

// Get window index from zone table
IF mZoneIndex > 0 AND mZoneIndex <= MAX_NUMBER_OF_ZONES THEN
	IF ZoneTable[mZoneIndex].TU_Present THEN
		mEndWindowIndex := ZoneTable[mZoneIndex].TU_EndWindowIndex;
	ELSE
		mNoTU_Available := TRUE;
		RETURN;
	END_IF
END_IF

// Check if window index was found
IF mEndWindowIndex > 0 THEN
	// Get position on tracking
	mPositionOnTracking := (TrackingPosition MOD TotalTrackingLength);
	
	IF WindowTable[mEndWindowIndex].TU_RearEdgePosition < mPositionOnTracking THEN
		M_GetTU_EndPosition := mPositionOnTracking - WindowTable[mEndWindowIndex].TU_RearEdgePosition;
	ELSE
		M_GetTU_EndPosition := mPositionOnTracking - WindowTable[mEndWindowIndex].TU_RearEdgePosition + TotalTrackingLength;
	END_IF
ELSE
	;// Window not found
END_IF
END_METHOD

/// Returns TU start position of a zone on tracked distance
/// Remark: User needs to make sure zone is valid
/// Remark: When no TU available the return value is 0, but is notfied with output "NoTuAvailable"
METHOD M_GetTU_StartPosition : UDINT // Start position of TU [mm]
VAR_INPUT
	mZoneIndex			: UINT; // Index of zone
END_VAR
VAR_OUTPUT
	mNoTU_Available		: BOOL; // No TU Available
END_VAR
VAR
	mStartWindowIndex	: UINT; // Zone end window index
	mPositionOnTracking	: UDINT; // Position on tracking length
END_VAR
M_GetTU_StartPosition := 0;
mStartWindowIndex := 0;
mNoTU_Available := FALSE;

// Get window index from zone table
IF mZoneIndex > 0 AND mZoneIndex <= MAX_NUMBER_OF_ZONES THEN
	IF ZoneTable[mZoneIndex].TU_Present THEN
		mStartWindowIndex := ZoneTable[mZoneIndex].TU_StartWindowIndex;
	ELSE
		mNoTU_Available := TRUE;
		RETURN;
	END_IF
END_IF

// Check if window index was found
IF mStartWindowIndex > 0 THEN
	// Get position on tracking
	mPositionOnTracking := (TrackingPosition MOD TotalTrackingLength);
	
	IF WindowTable[mStartWindowIndex].TU_FrontEdgePosition < mPositionOnTracking THEN
		M_GetTU_StartPosition := mPositionOnTracking - WindowTable[mStartWindowIndex].TU_FrontEdgePosition;
	ELSE
		M_GetTU_StartPosition := mPositionOnTracking - WindowTable[mStartWindowIndex].TU_FrontEdgePosition + TotalTrackingLength;
	END_IF
ELSE
	;// Window not found
END_IF
END_METHOD

/// Returns window index of an abolsute position
METHOD M_GetWindowIndex : UINT // Returns the Index of the Window if successful, otherwise 0 = No window
VAR_INPUT
	mAbsolutePosition	: UDINT; // Position on the tracking [mm]
END_VAR
VAR
	mTrackingPosition	: UDINT; // Current position on tracking
END_VAR
// Translate absolute position into position on tracking
mTrackingPosition := M_GetTrackingPosition(mAbsolutePosition);

IF WindowSize > 0 THEN
	M_GetWindowIndex := UDINT_TO_UINT(mTrackingPosition / WindowSize + 1);
ELSE
	M_GetWindowIndex := 0;
END_IF
END_METHOD

/// Returns position of Zone end on tracked distance
/// Remark: User needs to make sure zone is valid
METHOD M_GetZoneEndPosition : UDINT // Position of Zone end [mm]
VAR_INPUT
	mZoneIndex			: UINT; // Index of zone
END_VAR
VAR
	mEndWindowIndex		: UINT; // Zone end window index
	mPositionOnTracking	: UDINT; // Position on tracking length
END_VAR
M_GetZoneEndPosition := 0;
mEndWindowIndex := 0;

// Check inputs
IF mZoneIndex = 0 THEN
	RETURN;
END_IF

// Get window index from zone table
IF mZoneIndex > 0 AND mZoneIndex <= MAX_NUMBER_OF_ZONES THEN
	mEndWindowIndex := ZoneTable[mZoneIndex].ZoneEndWindowIndex;
END_IF

// Check if window index was found
IF mEndWindowIndex > 0 THEN
	// Get position on tracking
	mPositionOnTracking := (TrackingPosition MOD TotalTrackingLength);
	
	IF ZoneTable[mZoneIndex].ZoneEndPosition < mPositionOnTracking THEN
		M_GetZoneEndPosition := mPositionOnTracking - ZoneTable[mZoneIndex].ZoneEndPosition;
	ELSE
		M_GetZoneEndPosition := mPositionOnTracking - ZoneTable[mZoneIndex].ZoneEndPosition + TotalTrackingLength;
	END_IF
ELSE
	;// Window not found
END_IF
END_METHOD

/// Returns ZoneIndex at AbsolutePosition
METHOD M_GetZoneIndex : UINT // Returns ZoneIndex > 0, otherwise 0
VAR_INPUT
	mAbsolutePosition	: UDINT; // Position on the tracking [mm]
END_VAR
VAR
	mWindowIndex		: UINT; // Window index at position
	mZoneIndex			: UINT; // Zone index of window
	mTrackingPosition	: UDINT; // Abs position on tracking
END_VAR
M_GetZoneIndex := 0;

// Get window index of window position
mWindowIndex := M_GetWindowIndex(mAbsolutePosition);

// Return zone index
IF mWindowIndex > 0 AND mWindowIndex <= WindowTracking.MAX_NUMBER_OF_WINDOWS THEN
	mZoneIndex := WindowTable[mWindowIndex].ZoneIndex;
	
	IF mZoneIndex > 0 THEN
		mTrackingPosition := M_GetTrackingPosition(mAbsolutePosition);
		// When zone is allocated not over overflow position, range can be checked normally
		IF ZoneTable[mZoneIndex].ZoneEndPosition >= ZoneTable[mZoneIndex].ZoneStartPosition THEN
			// When requested tracking position is between start and end zone
			IF mTrackingPosition >= ZoneTable[mZoneIndex].ZoneStartPosition AND
			   mTrackingPosition <= ZoneTable[mZoneIndex].ZoneEndPosition THEN
			   M_GetZoneIndex := mZoneIndex;
			END_IF
			
		// When zone allocation is over overflow position, this needs to be considered
		ELSE
			// If request is between zone start and total tracking length
			IF mTrackingPosition >= ZoneTable[mZoneIndex].ZoneStartPosition THEN
				// Consider overflow and check range
				IF mTrackingPosition >= ZoneTable[mZoneIndex].ZoneStartPosition AND
				   mTrackingPosition <= (ZoneTable[mZoneIndex].ZoneStartPosition + ZoneTable[mZoneIndex].ZoneLength) THEN
				   M_GetZoneIndex := mZoneIndex;
				END_IF
				
			// Otherwise request was between tracking 0 to zone end
			ELSIF mTrackingPosition <= ZoneTable[mZoneIndex].ZoneEndPosition THEN
				// Correct request point upwards (Because of unsigned value)
				mTrackingPosition := mTrackingPosition + TotalTrackingLength;
			
				// Consider overflow and check range
				IF mTrackingPosition >= ZoneTable[mZoneIndex].ZoneStartPosition AND
				   mTrackingPosition <= (ZoneTable[mZoneIndex].ZoneStartPosition + ZoneTable[mZoneIndex].ZoneLength) THEN
				   M_GetZoneIndex := mZoneIndex;
				END_IF
			END_IF
		END_IF
	END_IF
END_IF
END_METHOD

/// Returns position of Zone start on tracked distance
/// Remark: User needs to make sure zone is valid
METHOD M_GetZoneStartPosition : UDINT // Position of Zone start [mm]
VAR_INPUT
	mZoneIndex			: UINT; // Index of zone
END_VAR
VAR
	mStartWindowIndex	: UINT; // Zone end window index
	mPositionOnTracking	: UDINT; // Position on tracking length
END_VAR
M_GetZoneStartPosition := 0;
mStartWindowIndex := 0;

// Check inputs
IF mZoneIndex = 0 THEN
	RETURN;
END_IF

// Get window index from zone table
IF mZoneIndex > 0 AND mZoneIndex <= MAX_NUMBER_OF_ZONES THEN
	mStartWindowIndex := ZoneTable[mZoneIndex].ZoneStartWindowIndex;
END_IF

// Check if window index was found
IF mStartWindowIndex > 0 THEN
	// Get position on tracking
	mPositionOnTracking := (TrackingPosition MOD TotalTrackingLength);
	
	IF ZoneTable[mZoneIndex].ZoneStartPosition < mPositionOnTracking THEN
		M_GetZoneStartPosition := mPositionOnTracking - ZoneTable[mZoneIndex].ZoneStartPosition;
	ELSE
		M_GetZoneStartPosition := mPositionOnTracking - ZoneTable[mZoneIndex].ZoneStartPosition + TotalTrackingLength;
	END_IF
ELSE
	;// Window not found
END_IF
END_METHOD

/// Inhibits shifting on a specific zone
METHOD M_InhibitShifting : BOOL // Returns true if successfully, otherwise false (e.g. Zone not found or not in use)
VAR_INPUT
	mZoneIndex		: UINT; // Zone index
	mInhibit		: BOOL; // True = Inhibit shifting
END_VAR
M_InhibitShifting := FALSE;

// Get window index from zone table
IF mZoneIndex > 0 AND mZoneIndex <= MAX_NUMBER_OF_ZONES THEN
	IF ZoneTable[mZoneIndex].Used THEN
		ZoneTable[mZoneIndex].InhibitShifting := mInhibit;
		M_InhibitShifting := TRUE;
	END_IF
END_IF
END_METHOD

// Initialize module - (e.g. calculates parameters)
// Remark: Does not delete anything on the tracking
METHOD M_Init : BOOL // Returns true if successful, otherwise false
VAR_INPUT
	mWindowSize				: UINT; // Size of windows [mm] Remark: Needs to be smaller than smallest transport unit
	mTrackingLength			: UDINT; // Length of tracking segment [mm] (e.g. conveyor length)
	mCurrentEncoderValue	: UDINT; // Current encoder value [inc]
	mMaxEncoderValueInc		: UDINT; // Max value of input "EncoderValue" [increments] Remark: Used to detect overflow
	mRateIncPerMM			: LREAL; // Ratio - How many increments represent one mm
	miEventListener			: I_WindowTrackingListener; // Tracking zone listener (0 = not used)
END_VAR
M_Init := FALSE;
Initialized := FALSE;

// Validate inputs
IF mWindowSize = 0 OR
   mTrackingLength = 0 OR 
   mRateIncPerMM = 0 OR 
   mMaxEncoderValueInc = 0 THEN
   RETURN;
END_IF

WindowSize := mWindowSize;
TrackingLength := mTrackingLength;
iEventListener := miEventListener;
RateIncPerMM := mRateIncPerMM;
MaxEncoderValueInc := mMaxEncoderValueInc;

TotalTrackingLength := M_CalculateTotalTrackingLength(
							 mTrackingLength 	:= TrackingLength,
							 mTrackingAddition 	:= TrackingAddition,
							 mWindowSize 		:= WindowSize);

MaxWindowIndex := UDINT_TO_UINT(TotalTrackingLength / WindowSize);

// Set start value
LastEncoderValueInc := mCurrentEncoderValue;

// Check window borders
IF MaxWindowIndex <= WindowTracking.MAX_NUMBER_OF_WINDOWS THEN
	Initialized := TRUE;						 
	M_Init := TRUE;
END_IF
END_METHOD

// Allocates a new zone slot and returns index
METHOD PROTECTED M_InsertNewZoneIndex : UINT // Returns zone index
VAR
	mIdx	: UINT; // Loop iterator
END_VAR
// Search free zone index
FOR mIdx := 1 TO MAX_NUMBER_OF_ZONES DO
	IF NOT ZoneTable[mIdx].Used THEN
		// Initialize Zone
		MEMSET(ADR(ZoneTable[mIdx]), 0, SIZEOF(ZoneTable[mIdx]));
		
		ZoneTable[mIdx].Used := TRUE;

		ZoneCount := ZoneCount + 1;	
	
		M_InsertNewZoneIndex := mIdx;
		RETURN;
	END_IF
END_FOR
END_METHOD

/// Checks wheter a shift is possible or not
METHOD PROTECTED M_IsShiftable : BOOL // Returns true if possible, otherwise false
VAR_INPUT
	mStartWindowIndex		: UINT; // Start window index of a zone to be shifted
	mWindowsToShift			: UINT; // Windows to shift
	mExcludeTUs				: BOOL; // Exclude physical occupied zones, otherwise shifting will fail due to a physical TU
	mAllowOverrun			: BOOL; // Allow to throw out zones which cannot be place on the tracking anymore because of reallocations
END_VAR
VAR_OUTPUT
	mZoneOverrun			: BOOL; // Overrun happening, zones availale which could not be placed on tracking
	mZoneOverrunWindowIndex	: UINT; // Window index where overrun started
END_VAR
VAR_IN_OUT
	mfbRelocator 			: FB_WindowRelocator; // Windows relocator
END_VAR
VAR_INST
	ResStartWindowIndex		: UINT; // Start window index where clean up starts
	MinShiftWindowIndex		: UINT; // Minimum window index until space has to be free 
	ResWindowsToShift		: UINT; // Result how many windows to be shifted 
	RemainingWindowLength 	: INT; // Remaining length on tracking, before reaching startpoint [windows]
	RelocScheduled 			: BOOL; // Reallocation processed successfully
	BlockingZoneIndex 		: UINT; // Index of a zone which was not permitted to be shifted (e.g. with physical TU inside)
	BlockingEndWindowIndex 	: UINT; // Last window index of blocking zone
	ErrorId 				: UINT; // Error id of reallocation process
	StartTrackingPosition	: UDINT; // Start position on tracking
	WindowsFromBegin		: UINT; // Amount of windows from beginning to the start position
	WindowsTrackingLength	: UINT; // Tracking length + Addition as windows
END_VAR
VAR
	mWindowIndex			: UINT; // Window index iterator
	mIdx 					: DINT; // Loop iterator
	mWindowLengthBlocking 	: UINT; // Length [windows] from start position to end of blocking zone
	mNextTargetWindow 		: UINT; // Next window index, where a Zone should be moved to
	mWindowLength 			: UINT; // Length [windows] of a zone
	mZoneIndexReloc 		: UINT; // Index of zone which should be reallocated
END_VAR
M_IsShiftable := FALSE;
mZoneOverrun := FALSE;
mZoneOverrunWindowIndex := 0;

// Validate inputs
IF mStartWindowIndex = 0 OR
   mStartWindowIndex > WindowTracking.MAX_NUMBER_OF_WINDOWS OR
   mWindowsToShift = 0 OR
   mWindowsToShift > WindowTracking.MAX_NUMBER_OF_WINDOWS OR
   WindowSize = 0 THEN
	RETURN;
END_IF

// Check start window index for an already available zone
// If there is one found align start window index to the start window index of this zone
IF WindowTable[mStartWindowIndex].ZoneIndex > 0 THEN
	ResStartWindowIndex := ZoneTable[WindowTable[mStartWindowIndex].ZoneIndex].ZoneStartWindowIndex;
ELSE
	ResStartWindowIndex := mStartWindowIndex;
END_IF

// Calculate minimum window index which has to be free 
//                  |-------------->
// Window     53 | 52 | 51 | 50 | 49
MinShiftWindowIndex := mStartWindowIndex + mWindowsToShift;
	
// Correct window border overflow
IF MinShiftWindowIndex > MaxWindowIndex THEN
	MinShiftWindowIndex := MinShiftWindowIndex - MaxWindowIndex;
END_IF

// Calculate windows which need to be shifted
// - From Startindex of Zone at Position X to the minimum distance to free
IF mStartWindowIndex >= ResStartWindowIndex THEN
	ResWindowsToShift := mWindowsToShift + mStartWindowIndex - ResStartWindowIndex;
ELSE
	ResWindowsToShift := mWindowsToShift + (mStartWindowIndex + MaxWindowIndex) - ResStartWindowIndex;
END_IF
	
// Go through all windows which need to be shifted mandatory
// and try to schedule a reallocation after the shifting distance.
mWindowIndex := ResStartWindowIndex;
mNextTargetWindow := MinShiftWindowIndex;
	
// Calculate available space on tracking which can be used for reallocations

// When zones get deleted on tracking end, the remaining distance to move reserved zones
// is limited to the windows up to the absolute window positions and the trackinglength backwards.
// Therefore from all windows of a TrackingLength - Startwindow is the distance 
// to be removed from the allowed shifting distance.
StartTrackingPosition := M_GetTrackingPosition((mStartWindowIndex-1)*WindowSize);
WindowsFromBegin := UDINT_TO_UINT(StartTrackingPosition / WindowSize);
WindowsTrackingLength := UDINT_TO_UINT((TrackingLength + TrackingAddition) / WindowSize);

IF WindowsFromBegin MOD WindowSize > 0 THEN
	WindowsFromBegin := WindowsFromBegin + 1;
END_IF

IF WindowsTrackingLength MOD WindowSize > 0 THEN
	WindowsTrackingLength := WindowsTrackingLength + 1;
END_IF

IF DeleteZoneTrackingEnd THEN	
	RemainingWindowLength := UINT_TO_INT(WindowsFromBegin) + UINT_TO_INT(WindowsTrackingLength) - UINT_TO_INT(ResWindowsToShift) - 1;
ELSE
	RemainingWindowLength := UINT_TO_INT(MaxWindowIndex) - UINT_TO_INT(ResWindowsToShift) - 1;
END_IF
	
FOR mIdx := 1 TO WindowTracking.MAX_NUMBER_OF_WINDOWS DO
	// Correct window border overflow
	IF mWindowIndex > MaxWindowIndex THEN
		mWindowIndex := mWindowIndex - MaxWindowIndex;
	END_IF
	
	IF mNextTargetWindow > MaxWindowIndex THEN
		mNextTargetWindow := mNextTargetWindow - MaxWindowIndex;
	END_IF
	
	// Relocation is done, if all zones in the shifting distance
	// and all interfering zones are relocated properly
	IF mIdx > ResWindowsToShift THEN
		M_IsShiftable := TRUE;
		EXIT;

	// If window is part of zone, try to schedule relocation
	ELSIF WindowTable[mWindowIndex].ZoneIndex > 0 THEN
		// Calculate Window Length of Zone which should be relocated
		mZoneIndexReloc := WindowTable[mWindowIndex].ZoneIndex;
		
		IF ZoneTable[mZoneIndexReloc].TU_Present THEN
			// Skip all occupied zones, because they are not allowed for re-allocation, otherwise fail
			IF mExcludeTUs THEN
				mWindowIndex := mWindowIndex + 1;
				RemainingWindowLength := RemainingWindowLength - 1;
				CONTINUE;
			ELSE
				M_IsShiftable := FALSE;
				EXIT;
			END_IF
		END_IF

		IF ZoneTable[mZoneIndexReloc].ZoneEndWindowIndex > ZoneTable[mZoneIndexReloc].ZoneStartWindowIndex THEN
			mWindowLength := ZoneTable[mZoneIndexReloc].ZoneEndWindowIndex - ZoneTable[mZoneIndexReloc].ZoneStartWindowIndex + 1;
		ELSE
			mWindowLength := ZoneTable[mZoneIndexReloc].ZoneEndWindowIndex + MaxWindowIndex  - ZoneTable[mZoneIndexReloc].ZoneStartWindowIndex + 1;
		END_IF

		// Check if reallocation would overwrite start point
		IF RemainingWindowLength - UINT_TO_INT(mWindowLength) > 0 THEN
			RelocScheduled := mfbRelocator.M_ScheduleRelocation(
									mZoneIndex				:= mZoneIndexReloc, 
									mTargetWindow			:= mNextTargetWindow, 
									mMaxWindowIndex			:= MaxWindowIndex, 
									mrWindowTable			:= WindowTable, 
									mrZoneTable				:= ZoneTable, 
									mBlockingZoneIndex		=> BlockingZoneIndex, 
									mBlockingEndWindowIndex => BlockingEndWindowIndex,
									mErrorId				=> ErrorId);
									
			// If relocation could be scheduled properly
			// set next window to the window after the relocated zone
			IF RelocScheduled THEN
				mNextTargetWindow := mNextTargetWindow + mWindowLength;
				
				// Adjust index of next window to check if relocation was successful
				mWindowIndex := mWindowIndex + mWindowLength;
				
				// Each found zone on the shifting distance requires one additional shift iteration
				// Because the location where it was moved to, may contains as well a zone which needs to be shifted
				ResWindowsToShift := ResWindowsToShift + 1;
				
				// Ensure that reallocation does not overwrite start point
				RemainingWindowLength := RemainingWindowLength - UINT_TO_INT(mWindowLength);
			ELSE
				// Relocation was not possible because of a Zone which is not allowed
				// to be shifted, try again with window after the blocking zone
				IF BlockingZoneIndex > 0 THEN
					// Each found zone on the shifting distance requires one additional shift iteration
					ResWindowsToShift := ResWindowsToShift + 1;
					
					// Calc length of blocking zone
					IF ZoneTable[BlockingZoneIndex].ZoneEndWindowIndex >= ZoneTable[BlockingZoneIndex].ZoneStartWindowIndex THEN
						mWindowLengthBlocking := ZoneTable[BlockingZoneIndex].ZoneEndWindowIndex - ZoneTable[BlockingZoneIndex].ZoneStartWindowIndex;
					ELSE
						mWindowLengthBlocking := ZoneTable[BlockingZoneIndex].ZoneEndWindowIndex + MaxWindowIndex - ZoneTable[BlockingZoneIndex].ZoneStartWindowIndex;
					END_IF
					
					mNextTargetWindow := BlockingEndWindowIndex + 1;
					
					RemainingWindowLength := RemainingWindowLength - UINT_TO_INT(mWindowLengthBlocking);
				END_IF
			END_IF
		ELSE
			// The found zone could not be placed on the tracking because there is no space left.
			// Mark overrun and leave
			mZoneOverrun := TRUE;
			mZoneOverrunWindowIndex := mWindowIndex;
			M_IsShiftable := mAllowOverrun;
			EXIT;
		END_IF
	ELSE
		mWindowIndex := mWindowIndex + 1;
		RemainingWindowLength := RemainingWindowLength - 1;
	END_IF
END_FOR
END_METHOD

/// Checks if a TU or a part of it, is found in a certain range.
METHOD M_IsTU_InRange : BOOL; // Returns true if present, otherwise false
VAR_INPUT
	mZoneIndex				: UINT; // Tracking zone index
	mAbsoluteStartRange		: UDINT; // Start range position on the tracking [mm]
	mAbsoluteEndRange		: UDINT; // End range position on the tracking [mm]
END_VAR
VAR
	mStartWindowIndex		: UINT; // Window index at start position
	mEndWindowIndex			: UINT; // Window index at end position
	mTrackingRangeEnd		: UDINT; // Tracking range position end
	mTrackingRangeStart		: UDINT; // Tracking range position start
	mTrackingTU_End			: UDINT; // Tracking range position end
	mTrackingTU_Start		: UDINT; // Tracking range position start
END_VAR
M_IsTU_InRange := FALSE;

// Check inputs
IF mZoneIndex = 0 THEN
	RETURN;
END_IF

IF NOT ZoneTable[mZoneIndex].TU_Present THEN
	RETURN;
END_IF

// Get window index of window start position
mStartWindowIndex := M_GetWindowIndex(mAbsoluteStartRange);
// Get window index of window end position
mEndWindowIndex := M_GetWindowIndex(mAbsoluteEndRange);

// Remark:
// Absolute view is unequal to tracking view
// ABS:  500mm 505mm .....1000mm
//   AbsStartpos		AbsEndPos
//       |                  |
//    TrackingEnd       TrackingStart
//
//  --------------------------------------      FlowDirection ->
// Win:  54  53  52 ....  43 42 ...
// Window index of end is normally lower than start (except overflow)     

// Ensure both window index are in a valid range
IF mStartWindowIndex > 0 AND mStartWindowIndex <= WindowTracking.MAX_NUMBER_OF_WINDOWS AND
   mEndWindowIndex > 0 AND mEndWindowIndex <= WindowTracking.MAX_NUMBER_OF_WINDOWS THEN
	
	// Ensure that Zone consists of start and end tu window index
	IF ZoneTable[mZoneIndex].TU_StartWindowIndex > 0 AND
	   ZoneTable[mZoneIndex].TU_EndWindowIndex > 0 THEN
	   
		//    TrackingEnd       TrackingStart
		//         |-----------------|
		//  --------------------------------------      FlowDirection ->
	   	mTrackingTU_End := WindowTable[ZoneTable[mZoneIndex].TU_EndWindowIndex].TU_RearEdgePosition;
	   	mTrackingTU_Start :=  WindowTable[ZoneTable[mZoneIndex].TU_StartWindowIndex].TU_FrontEdgePosition;
	   
		//    TrackingRangeEnd  TrackingRangeStart
		//      |----------------------|
		//  --------------------------------------      FlowDirection ->
		mTrackingRangeEnd := M_GetTrackingPosition(mAbsoluteStartRange);
   		mTrackingRangeStart := M_GetTrackingPosition(mAbsoluteEndRange);
	   
		// When range does not consists of the overflow point
		IF mTrackingRangeEnd >= mTrackingRangeStart THEN 
			// Check if TU End edge is between range
			IF mTrackingTU_End >= mTrackingRangeStart AND
               mTrackingTU_End <= mTrackingRangeEnd THEN
				M_IsTU_InRange := TRUE;
				RETURN;
				
			// Check if TU start edge is between range
			ELSIF mTrackingTU_Start >= mTrackingRangeStart AND
                  mTrackingTU_Start <= mTrackingRangeEnd THEN
				M_IsTU_InRange := TRUE;
				RETURN;
				
			// Check if TU is overlapping full range
			ELSIF mTrackingTU_End >= mTrackingRangeEnd AND
                  mTrackingTU_Start <= mTrackingRangeStart THEN
				M_IsTU_InRange := TRUE;
				RETURN; 
			END_IF
		// If range is overlapping overflow point
		ELSE
			// Check if TU End edge is between range
			IF mTrackingTU_End >= mTrackingRangeStart OR  
               mTrackingTU_End <= mTrackingRangeEnd THEN
				M_IsTU_InRange := TRUE;
				RETURN;
				
			// Check if TU start edge is between range
			ELSIF mTrackingTU_Start >= mTrackingRangeStart OR  
               mTrackingTU_Start <= mTrackingRangeEnd THEN
				M_IsTU_InRange := TRUE;
				RETURN;
				
			// Check if TU is overlapping full range
			ELSIF mTrackingTU_End >= mTrackingRangeEnd AND
                  mTrackingTU_Start <= mTrackingRangeStart THEN
				M_IsTU_InRange := TRUE;
				RETURN; 
			END_IF
		END_IF
	END_IF
END_IF
END_METHOD

/// Returns if a physical TU is present at mAbsolutePosition
METHOD M_IsTU_Present : BOOL; // Returns true if present, otherwise false
VAR_INPUT
	mAbsolutePosition		: UDINT; // Absolute position on tracking length
END_VAR
VAR
	mWindowIndex			: UINT; // Window index at absolute position
	mTrackingPosition		: UDINT; // Current position on tracking
END_VAR
M_IsTU_Present := FALSE;

// Get window index of position
mWindowIndex := M_GetWindowIndex(mAbsolutePosition);

IF mWindowIndex > 0 AND mWindowIndex <= WindowTracking.MAX_NUMBER_OF_WINDOWS THEN
	// Get position on tracking
	mTrackingPosition := M_GetTrackingPosition(mAbsolutePosition);

	// Get TU state
	CASE WindowTable[mWindowIndex].State OF
		E_WindowTrackingWindowState.IDLE:
			M_IsTU_Present := FALSE;
			
		E_WindowTrackingWindowState.FRONT_EDGE:
			IF WindowTable[mWindowIndex].TU_FrontEdgePosition <= mTrackingPosition THEN
				M_IsTU_Present := TRUE;
			ELSE
				M_IsTU_Present := FALSE;
			END_IF
		
		E_WindowTrackingWindowState.REAR_EDGE:
			IF WindowTable[mWindowIndex].TU_RearEdgePosition > mTrackingPosition THEN
				M_IsTU_Present := TRUE;
			ELSE
				M_IsTU_Present := FALSE;
			END_IF
		
		E_WindowTrackingWindowState.OCCUPIED:
			M_IsTU_Present := TRUE;
	END_CASE
END_IF
END_METHOD

/// Checks if a zone or a part of it,  is found in a certain range.
METHOD M_IsZoneInRange : BOOL; // Returns true if zone is in range, otherwise false
VAR_INPUT
	mZoneIndex				: UINT; // Tracking zone index
	mAbsoluteStartRange		: UDINT; // Start range position on the tracking [mm]
	mAbsoluteEndRange		: UDINT; // End range position on the tracking [mm]
END_VAR
VAR
	mStartWindowIndex		: UINT; // Window index at start position
	mEndWindowIndex			: UINT; // Window index at end position
	mTrackingRangeEnd		: UDINT; // Tracking range position end
	mTrackingRangeStart		: UDINT; // Tracking range position start
	mTrackingZoneEnd		: UDINT; // Tracking range position zone end
	mTrackingZoneStart		: UDINT; // Tracking range position zone start
END_VAR
M_IsZoneInRange := FALSE;

// Check inputs
IF mZoneIndex = 0 THEN
	RETURN;
END_IF

// Get window index of window start position
mStartWindowIndex := M_GetWindowIndex(mAbsoluteStartRange);
// Get window index of window end position
mEndWindowIndex := M_GetWindowIndex(mAbsoluteEndRange);

// Remark:
// Absolute view is unequal to tracking view
// ABS:  500mm 505mm .....1000mm
//    Startpos			 EndPos
//       |                  |
//  --------------------------------------      FlowDirection ->
// Win:  54  53  52 ....  43 42 ...
// Window index of end is normally lower than start (except overflow)     

// Ensure both window index are in a valid range
IF mStartWindowIndex > 0 AND mStartWindowIndex <= WindowTracking.MAX_NUMBER_OF_WINDOWS AND
   mEndWindowIndex > 0 AND mEndWindowIndex <= WindowTracking.MAX_NUMBER_OF_WINDOWS THEN

	// Ensure that Zone consists of start and end tu window index
	IF ZoneTable[mZoneIndex].TU_StartWindowIndex > 0 AND
	   ZoneTable[mZoneIndex].TU_EndWindowIndex > 0 THEN

		//    TrackingEnd       TrackingStart
		//         |-----------------|
		//  --------------------------------------      FlowDirection ->
	   	mTrackingZoneEnd := ZoneTable[mZoneIndex].ZoneEndPosition;
	   	mTrackingZoneStart := ZoneTable[mZoneIndex].ZoneStartPosition;

		//    TrackingRangeEnd  TrackingRangeStart
		//      |----------------------|
		//  --------------------------------------      FlowDirection ->
		mTrackingRangeEnd := M_GetTrackingPosition(mAbsoluteStartRange);
   		mTrackingRangeStart := M_GetTrackingPosition(mAbsoluteEndRange);

		// When range does not consists of the overflow point
		IF mTrackingRangeEnd >= mTrackingRangeStart THEN 
			// Check if TU End edge is between range
			IF mTrackingZoneEnd >= mTrackingRangeStart AND
               mTrackingZoneEnd <= mTrackingRangeEnd THEN
				M_IsZoneInRange := TRUE;
				RETURN;
				
			// Check if TU start edge is between range
			ELSIF mTrackingZoneStart >= mTrackingRangeStart AND
                  mTrackingZoneStart <= mTrackingRangeEnd THEN
				M_IsZoneInRange := TRUE;
				RETURN;
				
			// Check if TU is overlapping full range
			ELSIF mTrackingZoneEnd >= mTrackingRangeEnd AND
                  mTrackingZoneStart <= mTrackingRangeStart THEN
				M_IsZoneInRange := TRUE;
				RETURN; 
			END_IF
			
		// If range is overlapping overflow point
		ELSE
			// Check if TU End edge is between range
			IF mTrackingZoneEnd >= mTrackingRangeStart OR  
               mTrackingZoneEnd <= mTrackingRangeEnd THEN
				M_IsZoneInRange := TRUE;
				RETURN;
				
			// Check if TU start edge is between range
			ELSIF mTrackingZoneStart >= mTrackingRangeStart OR  
                  mTrackingZoneStart <= mTrackingRangeEnd THEN
				M_IsZoneInRange := TRUE;
				RETURN;
				
			// Check if TU is overlapping full range
			ELSIF mTrackingZoneEnd >= mTrackingRangeEnd AND
                  mTrackingZoneStart <= mTrackingRangeStart THEN
				M_IsZoneInRange := TRUE;
				RETURN; 
			END_IF
		END_IF
	END_IF
END_IF
END_METHOD

/// Tries to free a certain area by the following options (Shift, Shorten, Delete)
METHOD PROTECTED M_MakeSpace : BOOL // Returns true if successfully
VAR_INPUT
	mStartWindowIndex		: UINT; // Start window index
	mWindowsToFree			: UINT; // Windows to free up (e.g. 1 only clears start window index)
	mAllowZoneDelete		: BOOL; // Allows to delete zones if they could not be modified or reloacted
END_VAR
VAR_INST
	MinFreeWindowIndex		: UINT; // Minimum window index until space has to be free 
	ShiftZonesOk			: BOOL; // Shift was executed
END_VAR
VAR
	mIdx					: UINT; // Iteration
	mWindowIndex			: UINT; // Temp window index
	mZoneIndex				: UINT; // Zone index
	mTU_StartInArea			: BOOL; // TU start found in area
	mTU_EndInArea			: BOOL; // TU end found in area
END_VAR
// Initialize
M_MakeSpace := FALSE;

// Validate inputs
IF mStartWindowIndex = 0 OR
   mStartWindowIndex > WindowTracking.MAX_NUMBER_OF_WINDOWS OR
   mWindowsToFree = 0 OR
   mWindowsToFree > WindowTracking.MAX_NUMBER_OF_WINDOWS OR
   WindowSize = 0 THEN
	RETURN;
END_IF

// Initialize for-loop values
mWindowIndex := mStartWindowIndex;

// Calculate minimum window index which has to be free 
// Example: Startwindow 49, windows to be free 4 (49, 50, 51, 52)
//                  |-------------->
// Window     53 | 52 | 51 | 50 | 49
MinFreeWindowIndex := mStartWindowIndex + mWindowsToFree - 1;
	
// Correct window border overflow
IF MinFreeWindowIndex > MaxWindowIndex THEN
	MinFreeWindowIndex := MinFreeWindowIndex - MaxWindowIndex;
END_IF

// Check for any occupied zone in the area to be free and test if it spossible to shorten or delete it
FOR mIdx := 1 TO mWindowsToFree DO	
	IF WindowTable[mWindowIndex].ZoneIndex > 0 THEN
		mZoneIndex := WindowTable[mWindowIndex].ZoneIndex;
	
		// Zone can be modified by one of the following options
		// - If Occupied -> Shorten
		// - Else Delete if allowed
		IF ZoneTable[mZoneIndex].TU_Present THEN
			// Shorten
			// Check if position of TU inside the zone is outside of the area to be free
			IF MinFreeWindowIndex >= mStartWindowIndex THEN
				mTU_StartInArea := ZoneTable[mZoneIndex].TU_StartWindowIndex >= mStartWindowIndex AND
				   				   ZoneTable[mZoneIndex].TU_StartWindowIndex <= MinFreeWindowIndex;
				
				mTU_EndInArea := ZoneTable[mZoneIndex].TU_EndWindowIndex >= mStartWindowIndex AND
				   				 ZoneTable[mZoneIndex].TU_EndWindowIndex <= MinFreeWindowIndex;
				
			// Otherwise overflow between
			ELSE
				mTU_StartInArea := ZoneTable[mZoneIndex].TU_StartWindowIndex <= MinFreeWindowIndex OR
				   				   ZoneTable[mZoneIndex].TU_StartWindowIndex >= mStartWindowIndex;
				
				mTU_EndInArea := ZoneTable[mZoneIndex].TU_EndWindowIndex <= MinFreeWindowIndex OR
				   				 ZoneTable[mZoneIndex].TU_EndWindowIndex >= mStartWindowIndex;
			END_IF
			
			// TU Start or End is in area to be free
			IF mTU_StartInArea OR mTU_EndInArea THEN
				// Shorten not possible, check if delete is an option
				IF mAllowZoneDelete THEN
					// Ok
					;
				ELSE
					// Abort, shorten does not help
					M_MakeSpace := FALSE;
					RETURN;
				END_IF
			ELSE
				// Shorten is possible
				;
			END_IF
		END_IF
	END_IF
	
	mWindowIndex := mWindowIndex + 1;
	
	IF mWindowIndex > MaxWindowIndex THEN
		mWindowIndex := mWindowIndex - MaxWindowIndex;
	END_IF
END_FOR

// All occupied zones can be handled, try to shift 
ShiftZonesOk := M_ShiftZone(
					mStartWindowIndex,
					mWindowsToFree,
					TRUE,
					TRUE);

IF ShiftZonesOk THEN
	// First shorten zones at borders
	IF WindowTable[mStartWindowIndex].ZoneIndex > 0 THEN
		// If it consists of a TU
		IF ZoneTable[WindowTable[mStartWindowIndex].ZoneIndex].TU_Present THEN
			M_ShortenZoneAtWindow(
				WindowTable[mStartWindowIndex].ZoneIndex,
				mStartWindowIndex);
		END_IF
	END_IF

	IF WindowTable[MinFreeWindowIndex].ZoneIndex > 0 THEN
		// If it consists of a TU
		IF ZoneTable[WindowTable[MinFreeWindowIndex].ZoneIndex].TU_Present THEN
			M_ShortenZoneAtWindow(
				WindowTable[MinFreeWindowIndex].ZoneIndex,
				MinFreeWindowIndex);
		END_IF
	END_IF

	// Initialize loop
	mWindowIndex := mStartWindowIndex;
	
	// Execute TU operations
	FOR mIdx := 1 TO mWindowsToFree DO
		IF WindowTable[mWindowIndex].ZoneIndex > 0 THEN
			M_DeleteZone(WindowTable[mWindowIndex].ZoneIndex);
		END_IF
		
		mWindowIndex := mWindowIndex + 1;
	
		IF mWindowIndex > MaxWindowIndex THEN
			mWindowIndex := mWindowIndex - MaxWindowIndex;
		END_IF
	END_FOR
	
	M_MakeSpace := TRUE;
END_IF

IF NOT M_MakeSpace THEN
	// Error
	fbDebugMsg.M_SendErrorMsg('M_MakeSpace - Make space requested, but could not successfully executed.');	
END_IF
END_METHOD

/// Tries to free a certain area by the following options (Shift, Shorten, Delete)
METHOD PROTECTED M_MakeSpaceByWindows : BOOL // Returns true if successfully
VAR_INPUT
	mAbsolutePosition		: UDINT; // Start position window index
	mWindowsToFree			: UINT; // Windows to free up (e.g. 1 only clears start window index)
	mAllowZoneDelete		: BOOL; // Allows to delete zones if they could not be modified or reloacted
END_VAR

VAR
	mPositionWindowIndex	: UINT; // Window of position
END_VAR
M_MakeSpaceByWindows := FALSE;

// Validate inputs
IF WindowSize = 0 OR
   mWindowsToFree <= 0 THEN
	RETURN;
END_IF

mPositionWindowIndex := M_GetWindowIndex(mAbsolutePosition);

M_MakeSpaceByWindows := M_MakeSpace(
							mStartWindowIndex	:= mPositionWindowIndex, 
							mWindowsToFree		:= mWindowsToFree, 
							mAllowZoneDelete	:= mAllowZoneDelete);
END_METHOD

/// Allocates windows for ongoing transfers onto the belt 
/// until transfer gets completed by M_AddTU_RearEdge
/// Remark: Zones found during that process are tried to be shifted, otherwise deleted
METHOD PROTECTED M_ManageOngoingTransfers
VAR
	mIdx 				: UINT; // Loop iterator
	mWindowIndex		: UINT; // Current window iterator
	mTransferZoneIndex 	: UINT; // Transfer zone index iterator
	mFreeOk				: BOOL; // Shift ok
END_VAR
// Handle ongoing transfers onto the tracking belt
FOR mIdx := 1 TO TRANSFER_TABLE_SIZE DO
	// Check if dataset is active
	IF OngoingTransferList[mIdx].Active THEN
		// Get window index
		mWindowIndex := M_GetWindowIndex(OngoingTransferList[mIdx].AbsoluteInsertPosition);
		// Check if window has changed since last time
		IF mWindowIndex <> OngoingTransferList[mIdx].LastWindowIndex THEN
			IF mWindowIndex > 0 AND mWindowIndex <= WindowTracking.MAX_NUMBER_OF_WINDOWS THEN
				mTransferZoneIndex := OngoingTransferList[mIdx].ZoneIndex;
			
				// When a window gets overwritten which is already part of another zone, try to shift
				IF WindowTable[mWindowIndex].ZoneIndex > 0 AND
				   WindowTable[mWindowIndex].ZoneIndex <> mTransferZoneIndex THEN
					// Shift reserved zones
					mFreeOk := M_MakeSpaceByWindows(OngoingTransferList[mIdx].AbsoluteInsertPosition, 1, TRUE);
					
					// If not possible to shift, try to delete
					IF mFreeOk THEN
						DebugMsg := CONCAT('M_ManageOngoingTransfers - Could not free space. Zone: ',UINT_TO_STRING(WindowTable[mWindowIndex].ZoneIndex));
						fbDebugMsg.M_SendInfoMsg(DebugMsg);
					END_IF
				END_IF
				
				// A zone index needs to be available
				IF mTransferZoneIndex > 0 THEN
					// Update zone as currently end of TU, even this is not the last window to ensure always valid zone configuration
					// Otherwise it is unclear how many windows are part of a zone.
					WindowTable[mWindowIndex].State := E_WindowTrackingWindowState.REAR_EDGE;
					WindowTable[mWindowIndex].TU_RearEdgePosition := mWindowIndex * WindowSize - 1;
					
					WindowTable[mWindowIndex].ZoneIndex := OngoingTransferList[mIdx].ZoneIndex;
					ZoneTable[mTransferZoneIndex].ZoneEndWindowIndex := mWindowIndex;
					ZoneTable[mTransferZoneIndex].TU_EndWindowIndex := mWindowIndex;
					ZoneTable[mTransferZoneIndex].ZoneEndPosition := mWindowIndex * WindowSize - 1;
					
					
					IF ZoneTable[mTransferZoneIndex].ZoneEndPosition >= ZoneTable[mTransferZoneIndex].ZoneStartPosition THEN
						ZoneTable[mTransferZoneIndex].ZoneLength := UDINT_TO_UINT(ZoneTable[mTransferZoneIndex].ZoneEndPosition 
																				   - ZoneTable[mTransferZoneIndex].ZoneStartPosition);
					ELSE
						ZoneTable[mTransferZoneIndex].ZoneLength := UDINT_TO_UINT(ZoneTable[mTransferZoneIndex].ZoneEndPosition 
																				  + TotalTrackingLength 
																				  - ZoneTable[mTransferZoneIndex].ZoneStartPosition);
					END_IF
					
					// When a last is available (Was last rear edge, update to occupied 
					IF OngoingTransferList[mIdx].LastWindowIndex > 0 THEN
						IF WindowTable[OngoingTransferList[mIdx].LastWindowIndex].State = E_WindowTrackingWindowState.REAR_EDGE THEN
							WindowTable[OngoingTransferList[mIdx].LastWindowIndex].State := E_WindowTrackingWindowState.OCCUPIED;
							WindowTable[OngoingTransferList[mIdx].LastWindowIndex].TU_RearEdgePosition := 0;
						END_IF
					END_IF
					
					// Update transfer list
					OngoingTransferList[mIdx].LastWindowIndex := mWindowIndex;
				ELSE
					// Error
					;
				END_IF
			END_IF
		END_IF	
	ELSE
		EXIT;
	END_IF
END_FOR
END_METHOD

/// Monitors if one of the registered zones reach PTL, so they can be deleted
METHOD PROTECTED M_MonitorZonesPTL
VAR
	mIdx 				: UINT; // Loop iterator
	mPosition			: UDINT; // Current zone end position
END_VAR
// Handle ongoing ptl on the tracking distance
FOR mIdx := 1 TO MAX_NUMBER_OF_ZONES DO
	// Check if dataset is active
	IF PTL_Zones[mIdx] > 0 THEN		
		mPosition := M_GetZoneEndPosition(PTL_Zones[mIdx]);
		
		// Zone which consists of a TU or which are not valid anymore
		// get deleted from list, so they are not monitored anymore
		IF NOT ZoneTable[PTL_Zones[mIdx]].Used OR
		   ZoneTable[PTL_Zones[mIdx]].TU_Present THEN
			M_RemoveZoneFromPTL(PTL_Zones[mIdx]);
			
		// When the absolute position of zone end is reached, delete zone
		ELSIF mPosition > ZoneTable[PTL_Zones[mIdx]].PositionToLive AND mPosition < ZoneTable[PTL_Zones[mIdx]].PositionToLive + TrackingLength THEN
			M_DeleteZone(PTL_Zones[mIdx]);
		END_IF
	ELSE
		EXIT;
	END_IF
END_FOR
END_METHOD

/// Moves all windows of a zone to another target window. (Possible edges are applied as before in the new window)
/// Remark: Possible zones at destination get shifted or deleted based on configuration if possible.
METHOD PROTECTED M_MoveZone : BOOL // Returns true if successfully moved, otherwise false (e.g. target consists of a non movable zone)
VAR_INPUT
	mZoneIndex				: UINT; // Zone index to move
	mTargetStartWindow 		: UINT; // Target start window index
	mEnableDeleteOfZones  	: BOOL; // Zones at target destination gets deleted if they can not be shifted or shortened
END_VAR

VAR
	mIdx 					: UINT; // Loop iterator
	mZoneWindowLength 		: UINT; // Length of zone to be moved
	mWindowIndex 			: UINT; // Iterator window index loop
	mBufferOk				: BOOL; // Command executed successfully
END_VAR

VAR_INST
	MovePossible			: BOOL;
	OldRelWindowPositionRE 	: UDINT; // Old relative window position rear edge
	OldRelWindowPositionFE 	: UDINT; // Old relative window position front edge
	OldRelZoneStartPosition : UDINT; // Old relative zone start position
	OldRelZoneEndPosition 	: UDINT; // Old relative zone end position
	fbWindowBuffer			: FB_MemRingBuffer; // Temporary storage of source windows
	WindowBuffer			: ARRAY[1..(MAX_MOVE_WINDOWS * SIZEOF(ST_WindowTrackingWindow))] OF BYTE; // Buffer storage
END_VAR
M_MoveZone := FALSE;

// Validate inputs
IF mZoneIndex <= 0 OR
   mZoneIndex > MAX_NUMBER_OF_ZONES OR
   mTargetStartWindow = 0 OR
   mTargetStartWindow > MaxWindowIndex  THEN
   RETURN;
END_IF

// Calculate length of zone to move [windows]
IF ZoneTable[mZoneIndex].ZoneEndWindowIndex > ZoneTable[mZoneIndex].ZoneStartWindowIndex THEN
	mZoneWindowLength := ZoneTable[mZoneIndex].ZoneEndWindowIndex - ZoneTable[mZoneIndex].ZoneStartWindowIndex + 1;
ELSE
	mZoneWindowLength := ZoneTable[mZoneIndex].ZoneEndWindowIndex + MaxWindowIndex - ZoneTable[mZoneIndex].ZoneStartWindowIndex + 1;
END_IF


mWindowIndex := mTargetStartWindow;
MovePossible := TRUE;

IF NOT mEnableDeleteOfZones THEN
	// Clear target
	FOR mIdx := 1 TO mZoneWindowLength DO
		// Check if target is free or already part of the same zone
		IF WindowTable[mWindowIndex].ZoneIndex > 0 AND
		   WindowTable[mWindowIndex].ZoneIndex <> mZoneIndex THEN
		   
			// Make sure destination is free
			MovePossible := M_MakeSpace(
								mWindowIndex,
								1,
								mEnableDeleteOfZones);
								
			IF NOT MovePossible THEN
				EXIT;
			END_IF
		END_IF
		
		mWindowIndex := mWindowIndex + 1;
			
		// Correct border overflow
		IF mWindowIndex > MaxWindowIndex THEN
			mWindowIndex := mWindowIndex - MaxWindowIndex;
		END_IF
	END_FOR
END_IF

// When target is clear to receive a zone
IF MovePossible THEN
	// Clear temporary window buffer
	fbWindowBuffer.A_Reset(
		pBuffer 	:= ADR(WindowBuffer), 
		cbBuffer 	:= SIZEOF(WindowBuffer));
	
	mWindowIndex := ZoneTable[mZoneIndex].ZoneStartWindowIndex; 
	
	// Source windows needs to be stored temporarly, because it is possible
	// that the new target is inside the existing window range.
	FOR mIdx := 1 TO mZoneWindowLength DO
		// Add existing window to buffer
		fbWindowBuffer.A_AddTail(
			pBuffer 	:= ADR(WindowBuffer), 
			cbBuffer 	:= SIZEOF(WindowBuffer), 
			pWrite 		:= ADR(WindowTable[mWindowIndex]), 
			cbWrite 	:= SIZEOF(WindowTable[mWindowIndex]));
			
		mBufferOk := fbWindowBuffer.bOk;
			
		// Clear source window
		M_ClearWindow(mWindowIndex);
		
		mWindowIndex := mWindowIndex + 1;
		
		// Correct border overflow
		IF mWindowIndex > MaxWindowIndex THEN
			mWindowIndex := mWindowIndex - MaxWindowIndex;
		END_IF
	END_FOR
	
	// Copy source window to destination and update zone information
	mWindowIndex := mTargetStartWindow;
	
	FOR mIdx := 1 TO mZoneWindowLength DO
		// Copy window by window to target
		fbWindowBuffer.A_RemoveHead(
			pBuffer 	:= ADR(WindowBuffer), 
			cbBuffer 	:= SIZEOF(WindowBuffer), 
			pRead 		:= ADR(WindowTable[mWindowIndex]), 
			cbRead 		:= SIZEOF(WindowTable[mWindowIndex]));
		
		mBufferOk := fbWindowBuffer.bOk;
		
		// Update begin and end of zone
		IF mIdx = 1 THEN
			ZoneTable[mZoneIndex].ZoneStartWindowIndex := mWindowIndex;
			
		ELSIF mIdx = mZoneWindowLength THEN
			ZoneTable[mZoneIndex].ZoneEndWindowIndex := mWindowIndex;
		END_IF
		
		// When the moved window is marked as Front edge, update zone and position based on new window
		IF WindowTable[mWindowIndex].State = E_WindowTrackingWindowState.FRONT_EDGE THEN
			ZoneTable[mZoneIndex].TU_StartWindowIndex := mWindowIndex;
			OldRelWindowPositionFE := WindowTable[mWindowIndex].TU_FrontEdgePosition MOD WindowSize;
			WindowTable[mWindowIndex].TU_FrontEdgePosition := OldRelWindowPositionFE + (mWindowIndex-1) * WindowSize;
			
		// When the moved window is marked as Rear edge, update zone and position based on new window	
		ELSIF WindowTable[mWindowIndex].State = E_WindowTrackingWindowState.REAR_EDGE THEN 
			ZoneTable[mZoneIndex].TU_EndWindowIndex := mWindowIndex;
			OldRelWindowPositionRE := WindowTable[mWindowIndex].TU_RearEdgePosition MOD WindowSize;
			WindowTable[mWindowIndex].TU_RearEdgePosition := OldRelWindowPositionRE + (mWindowIndex-1) * WindowSize;
		END_IF
		
		mWindowIndex := mWindowIndex + 1;
		
		// Correct border overflow
		IF mWindowIndex > MaxWindowIndex THEN
			mWindowIndex := mWindowIndex - MaxWindowIndex;
		END_IF
	END_FOR
	
	// Update zone start and end position to new windows
	OldRelZoneStartPosition := ZoneTable[mZoneIndex].ZoneStartPosition MOD WindowSize;
	OldRelZoneEndPosition := ZoneTable[mZoneIndex].ZoneEndPosition MOD WindowSize;
	
	ZoneTable[mZoneIndex].ZoneStartPosition := OldRelZoneStartPosition + (ZoneTable[mZoneIndex].ZoneStartWindowIndex-1) * WindowSize;
	ZoneTable[mZoneIndex].ZoneEndPosition := OldRelZoneEndPosition + (ZoneTable[mZoneIndex].ZoneEndWindowIndex-1) * WindowSize;
	
	// Inform listener
	IF iEventListener <> 0 THEN
		iEventListener.M_TrackingZoneMovedEvent(
			mTrackingZoneIndex 	:= mZoneIndex,
			mTrackingZoneData 	:= ZoneTable[mZoneIndex]);
	END_IF
	
	M_MoveZone := TRUE;
END_IF
END_METHOD

/// Moves all windows of a zone to another target window aligned on front edge.
/// Remark: Possible zones at destination get shifted or deleted based on configuration.
/// Remark: If a physical TU can be found at Target, move not possible
METHOD PROTECTED M_MoveZoneFE : BOOL // Returns true if successful moved, otherwise false 
VAR_INPUT
	mZoneIndex					: UINT; // Zone index to move
	mAbsoluteTargetPosition		: UDINT; // Absolute target position [mm]
	mDeleteTargetZones  		: BOOL; // Zones at target destination gets deleted, otherwise shifted
END_VAR

VAR
	mMoveOk						: BOOL; // Move to new window location was successful
	mFrontEdgeAdjusted			: BOOL; // Front edge successfull adjusted
END_VAR

VAR_INST
	WindowNumberFE 				: UINT; // Number of front edge window in zone
	TargetWindowIndex			: UINT; // Target window index
	TargetMoveWindowIndex		: UINT; // Target move window index
	ZoneWindowLength 			: UINT; // Length of zone to be moved
	EdgeWindowIndex				: UINT; // Edge window index of zone
	NewTrackingPosition			: UDINT; // New required tracking position
	OldZoneStartWindowIndex 	: UINT; // Old zone start window index (Rollback)
END_VAR
M_MoveZoneFE := FALSE;

// Validate inputs
IF mZoneIndex <= 0 OR
   mZoneIndex > MAX_NUMBER_OF_ZONES OR
   WindowSize = 0 THEN
   RETURN;
END_IF

// Get window index of target position
TargetWindowIndex := M_GetWindowIndex(mAbsoluteTargetPosition);
   
// Ensure window is valid and physically occupied
IF ZoneTable[mZoneIndex].TU_Present AND
   TargetWindowIndex > 0 AND TargetWindowIndex <= WindowTracking.MAX_NUMBER_OF_WINDOWS THEN
   
	// Calculate length of zone in windows
	IF ZoneTable[mZoneIndex].ZoneEndWindowIndex > ZoneTable[mZoneIndex].ZoneStartWindowIndex THEN
		ZoneWindowLength := ZoneTable[mZoneIndex].ZoneEndWindowIndex - ZoneTable[mZoneIndex].ZoneStartWindowIndex + 1;
	ELSE
		ZoneWindowLength := ZoneTable[mZoneIndex].ZoneEndWindowIndex + MaxWindowIndex  - ZoneTable[mZoneIndex].ZoneStartWindowIndex + 1;
	END_IF
	
	// Store front edge and position of it in zone
	EdgeWindowIndex := ZoneTable[mZoneIndex].TU_StartWindowIndex;
	
	IF EdgeWindowIndex >= ZoneTable[mZoneIndex].ZoneStartWindowIndex THEN
		WindowNumberFE := EdgeWindowIndex - ZoneTable[mZoneIndex].ZoneStartWindowIndex + 1;
	ELSE
		WindowNumberFE := EdgeWindowIndex + MaxWindowIndex - ZoneTable[mZoneIndex].ZoneStartWindowIndex + 1;
	END_IF
	
	// If an edge is available
	IF EdgeWindowIndex > 0 THEN
		IF TargetWindowIndex >= WindowNumberFE THEN
			TargetMoveWindowIndex := TargetWindowIndex - WindowNumberFE + 1;
		ELSE
			TargetMoveWindowIndex := TargetWindowIndex + MaxWindowIndex - WindowNumberFE + 1;
		END_IF
		
		// Store old window index for a possible rollback
		OldZoneStartWindowIndex := ZoneTable[mZoneIndex].ZoneStartWindowIndex;
		
		// Move zone to target
		mMoveOk := M_MoveZone(
						mZoneIndex 				:= mZoneIndex,
						mTargetStartWindow 		:= TargetMoveWindowIndex,
						mEnableDeleteOfZones 	:= FALSE);	
		
		// If zone could be moved to new location, 
		IF mMoveOk THEN
			NewTrackingPosition := M_GetTrackingPosition(mAbsoluteTargetPosition);
			
			// try to adapt edge position changes (Front edge and rear edge)
			mFrontEdgeAdjusted := M_AdjustFE(
									mWindowIndexFE 			:= TargetWindowIndex,
									mNewTrackingPosition 	:= NewTrackingPosition,
									mDeleteTargetZones 		:= mDeleteTargetZones);
		
			IF mFrontEdgeAdjusted THEN
				// Move successful
				M_MoveZoneFE := TRUE;
			
			// Edge could not be aligned -> Rollback and abort		
			ELSE
				mMoveOk := M_MoveZone(
							mZoneIndex 				:= mZoneIndex,
							mTargetStartWindow 		:= OldZoneStartWindowIndex,
							mEnableDeleteOfZones 	:= FALSE);
							
				IF NOT mMoveOk THEN
					// Error during rollback
					;
				END_IF
				
				M_MoveZoneFE := FALSE;
			END_IF		
											
		// Move was not possible -> Abort						
		ELSE
			M_MoveZoneFE := FALSE;
		END_IF	
		
	// Otherwise no front edge window found
	ELSE
		M_MoveZoneFE := FALSE;
	END_IF
// Zone not valid 
ELSE
	M_MoveZoneFE := FALSE;
END_IF
END_METHOD

/// Moves all windows of a zone to another target window aligned on rear edge.
/// Remark: Possible zones at destination get shifted or deleted based on configuration.
/// Remark: If a physical TU can be found at Target, move not possible
METHOD PROTECTED M_MoveZoneRE : BOOL // Returns true if successful moved, otherwise false 
VAR_INPUT
	mZoneIndex					: UINT; // Zone index to move
	mAbsoluteTargetPosition		: UDINT; // Absolute target position [mm]
	mDeleteTargetZones  		: BOOL; // Zones at target destination gets deleted, otherwise shifted
END_VAR

VAR
	mMoveOk						: BOOL; // Move to new window location was successful
	mRearEdgeAdjusted			: BOOL; // Rear edge adjusted successfully
END_VAR

VAR_INST
	TargetWindowIndex			: UINT; // Target window index
	TargetMoveWindowIndex		: UINT; // Target move window index
	ZoneWindowLength 			: UINT; // Length of zone to be moved
	EdgeWindowIndex				: UINT; // Edge window index of zone
	WindowNumberRE 				: UINT; // Number of window in zone
	NewTrackingPosition			: UDINT; // new required tracking position
	OldZoneStartWindowIndex 	: UINT; // Old zone start window index (Rollback)
END_VAR
M_MoveZoneRE := FALSE;

// Validate inputs
IF mZoneIndex <= 0 OR
   mZoneIndex > MAX_NUMBER_OF_ZONES OR
   WindowSize = 0 THEN
   RETURN;
END_IF

// Get window index of target position
TargetWindowIndex := M_GetWindowIndex(mAbsoluteTargetPosition);
   
// Ensure window is valid and physically occupied
IF ZoneTable[mZoneIndex].TU_Present AND
   TargetWindowIndex > 0 AND TargetWindowIndex <= WindowTracking.MAX_NUMBER_OF_WINDOWS THEN 
	// Calculate length of zone in windows
	IF ZoneTable[mZoneIndex].ZoneEndWindowIndex > ZoneTable[mZoneIndex].ZoneStartWindowIndex THEN
		ZoneWindowLength := ZoneTable[mZoneIndex].ZoneEndWindowIndex - ZoneTable[mZoneIndex].ZoneStartWindowIndex + 1;
	ELSE
		ZoneWindowLength := ZoneTable[mZoneIndex].ZoneEndWindowIndex + MaxWindowIndex  - ZoneTable[mZoneIndex].ZoneStartWindowIndex + 1;
	END_IF
	
	// Store rear edge and position of it in zone
	EdgeWindowIndex := ZoneTable[mZoneIndex].TU_EndWindowIndex;
	
	IF EdgeWindowIndex >= ZoneTable[mZoneIndex].ZoneEndWindowIndex THEN
		WindowNumberRE := EdgeWindowIndex - ZoneTable[mZoneIndex].ZoneEndWindowIndex + 1;
	ELSE
		WindowNumberRE := EdgeWindowIndex + MaxWindowIndex - ZoneTable[mZoneIndex].ZoneEndWindowIndex + 1;
	END_IF
	
	// If an rear edge was found
	IF EdgeWindowIndex > 0 THEN
		// Calculate offset to ensure that rear edge window is at target window after move operation
		IF TargetWindowIndex >= WindowNumberRE THEN
			TargetMoveWindowIndex := TargetWindowIndex - WindowNumberRE + 1;
		ELSE
			TargetMoveWindowIndex := TargetWindowIndex + MaxWindowIndex - WindowNumberRE + 1;
		END_IF
		
		// Store old window index for a possible rollback
		OldZoneStartWindowIndex := ZoneTable[mZoneIndex].ZoneStartWindowIndex;

		// Move zone to target 
		mMoveOk := M_MoveZone(
						mZoneIndex 				:= mZoneIndex,
						mTargetStartWindow 		:= TargetMoveWindowIndex,
						mEnableDeleteOfZones 	:= FALSE);	
		
		// If zone could be moved to new location, 
		IF mMoveOk THEN
			NewTrackingPosition := M_GetTrackingPosition(mAbsoluteTargetPosition);
			
			// try to adapt edge position changes (Front edge and rear edge)
			mRearEdgeAdjusted := M_AdjustRE(
									mWindowIndexRE 			:= TargetWindowIndex,
									mNewTrackingPosition 	:= NewTrackingPosition,
									mDeleteTargetZones 		:= mDeleteTargetZones);
		
			IF mRearEdgeAdjusted THEN
				// Move successful
				M_MoveZoneRE := TRUE;
			
			// Edge could not be aligned -> Rollback and abort		
			ELSE
				fbDebugMsg.M_SendErrorMsg('M_MoveZoneRE - Rear edge could no be adjusted.');	
			
				mMoveOk := M_MoveZone(
							mZoneIndex 				:= mZoneIndex,
							mTargetStartWindow 		:= OldZoneStartWindowIndex,
							mEnableDeleteOfZones 	:= FALSE);
							
				IF NOT mMoveOk THEN
					// Error during rollback
					fbDebugMsg.M_SendErrorMsg('M_MoveZoneRE - Rollback not possible.');	
				END_IF
				
				M_MoveZoneRE := FALSE;
			END_IF
												
		// Move was not possible -> Abort						
		ELSE
			M_MoveZoneRE := FALSE;
		END_IF
		
	// Otherwise no rear edge window found
	ELSE
		M_MoveZoneRE := FALSE;
	END_IF
// Zone not valid 
ELSE
	M_MoveZoneRE := FALSE;
END_IF
END_METHOD

/// Removes a zone from the ptl list and closes all gaps in list
METHOD PROTECTED M_RemoveZoneFromPTL : BOOL // Returns true if zone was found and deleted, otherwise false
VAR_INPUT
	mZoneIndex			: UINT; // Zone index to remove
END_VAR
VAR
	mIdx				: UINT; // Iterator
	mCloseGapsInList 	: BOOL; // Flag to close gaps
END_VAR
M_RemoveZoneFromPTL := FALSE;
mCloseGapsInList := FALSE;

// Clean entry in PTL list and close gaps in list
FOR mIdx := 1 TO MAX_NUMBER_OF_ZONES DO
	IF PTL_Zones[mIdx] <> 0  THEN	
		IF PTL_Zones[mIdx] = mZoneIndex THEN 
			// Clear entry and mark following to close gaps
			mCloseGapsInList := TRUE;
			PTL_Zones[mIdx] := 0;
			M_RemoveZoneFromPTL := TRUE;
			
		ELSIF mCloseGapsInList THEN
			// Close gaps
			PTL_Zones[mIdx-1] := PTL_Zones[mIdx];
			PTL_Zones[mIdx] := 0;
		END_IF
	ELSE
		// No entries available
		EXIT;
	END_IF
END_FOR
END_METHOD

/// Removes a zone from the transfer list and closes all gaps in list
METHOD PROTECTED M_RemoveZoneFromTransferList : BOOL // Returns true if zone was found and deleted, otherwise false
VAR_INPUT
	mZoneIndex			: UINT; // Zone index to remove
END_VAR
VAR
	mIdx				: UINT; // Iterator
	mCloseGapsInList 	: BOOL; // Flag to close gaps
END_VAR
M_RemoveZoneFromTransferList := FALSE;
mCloseGapsInList := FALSE;

// Clean entry in transfer list and close gaps in list
FOR mIdx := 1 TO TRANSFER_TABLE_SIZE DO
	IF OngoingTransferList[mIdx].Active THEN	
		IF OngoingTransferList[mIdx].ZoneIndex = mZoneIndex THEN 
			// Clear entry and mark following to close gaps
			mCloseGapsInList := TRUE;
			MEMSET(ADR(OngoingTransferList[mIdx]), 0, SIZEOF(OngoingTransferList[mIdx]));
			M_RemoveZoneFromTransferList := TRUE;
			
		ELSIF mCloseGapsInList THEN
			// Close gaps
			OngoingTransferList[mIdx-1] := OngoingTransferList[mIdx];
			MEMSET(ADR(OngoingTransferList[mIdx]), 0, SIZEOF(OngoingTransferList[mIdx]));
		END_IF
	ELSE
		// No entries available
		EXIT;
	END_IF
END_FOR
END_METHOD

/// Reserve a Zone on tracking
/// Remark: Target needs to be free
METHOD PROTECTED M_ReserveZone : UINT // Returns Zone index if successful, otherwise 0
VAR_INPUT
	mActionId						: INT; (* ID of action which requests zone - 
								     		(0 = Only reservation, but free to be used by other actions) *)
	mLength							: UINT; // Length of zone to allocate [mm]
	mStartWindowIndex 				: UINT; // Start window index
	mStartTrackingPosition			: UDINT; // Start tracking position of the zone in start window [mm]
	mInhibitShifting				: BOOL; // Mark zone as not shiftable
	miActionListener				: I_TrackingActionListener; // Action listener of the created zone
	mPositionToLive					: UDINT; // Absolute position until allocation gets deleted automatically if not used (0 = disabled)
END_VAR
VAR_INST
	ZoneIndex 						: UINT; // Allocated zone index
	MaxWindowPosition 				: UDINT; // Input check for required poition MAX
	MinWindowPosition 				: UDINT; // Input check for required poition MIN
END_VAR
VAR
	mIdx							: UINT; // Loop iterator
	mWindowIndex					: UINT; // Start window index
	mWindowLength					: UINT; // Zone length in windows
	mEndWindowIndex					: UINT; // End window index
	mReservationAllowed 			: BOOL; // Reservation valid (e.g. free space available)
	mZoneEndPosition				: UDINT; // Zone end position 
	mRelWindowPositionZoneStart 	: UDINT; // Relative position of zone start in window
	mFullLength						: UINT; // Full length to be allocated
END_VAR
M_ReserveZone := 0;

// Validate inputs
IF mLength <= 0 OR
   WindowSize = 0 OR
   mStartWindowIndex <= 0 OR
   mStartWindowIndex > WindowTracking.MAX_NUMBER_OF_WINDOWS THEN
   RETURN;
END_IF

// Get max and min tracking position of front edge window
MaxWindowPosition := (mStartWindowIndex) * WindowSize;
MinWindowPosition := (mStartWindowIndex-1) * WindowSize;

// Ensure that new tracking position is in range of window
IF mStartTrackingPosition < MinWindowPosition OR 
   mStartTrackingPosition >= MaxWindowPosition THEN
   RETURN;
END_IF

// Calculate relative position in first zone window
mRelWindowPositionZoneStart := mStartTrackingPosition MOD WindowSize;

// The relative position in the first window is added to the length, 
// in order to get the amount of windows which are allocated for that TU finally
mFullLength := mLength + UDINT_TO_UINT(mRelWindowPositionZoneStart);

// Convert length into number of windows
mWindowLength := mFullLength / WindowSize;
// If not the full length could be mapped in windows
// add an additional window
IF (mFullLength MOD WindowSize) > 0 THEN
	mWindowLength := mWindowLength + 1;
END_IF

mWindowIndex := mStartWindowIndex;
mReservationAllowed := TRUE;

// Ensure reservation is possible
FOR mIdx := 1 TO mWindowLength DO
	// When zone is not empty or marked as flush, abort
	IF WindowTable[mWindowIndex].ZoneIndex > 0  OR
	   WindowTable[mWindowIndex].Flush THEN
	   // Cancel resevation
	   mReservationAllowed := FALSE;
	   M_ReserveZone := 0;
	   
	   	// Error
		fbDebugMsg.M_SendErrorMsg('M_ReserveZone - Reservation not possible, no available space.');	
	   	RETURN;
	END_IF
	
	mWindowIndex := mWindowIndex + 1;
 
	// Correct border overflow
	IF mWindowIndex > MaxWindowIndex THEN
		mWindowIndex := mWindowIndex - MaxWindowIndex;
	END_IF
END_FOR

// When reservation is possible to be executed
IF mReservationAllowed THEN
	// Get new Zone index
	ZoneIndex := M_InsertNewZoneIndex();
	
	IF ZoneIndex > 0 THEN
		mWindowIndex := mStartWindowIndex;
		
		// Loop through all windows and assigne new zone
		FOR mIdx := 1 TO mWindowLength DO
		   // Clear window
			MEMSET(ADR(WindowTable[mWindowIndex]),0,SIZEOF(WindowTable[mWindowIndex]));
			
			WindowTable[mWindowIndex].ZoneIndex := ZoneIndex;
			WindowTable[mWindowIndex].State := E_WindowTrackingWindowState.RESERVED;
							
			mWindowIndex := mWindowIndex + 1;
		 
			// Correct border overflow
			IF mWindowIndex > MaxWindowIndex THEN
				mWindowIndex := mWindowIndex - MaxWindowIndex;
			END_IF
		END_FOR
		
		mEndWindowIndex := mStartWindowIndex + mWindowLength - 1;
		
		// Correct border overflow
		IF mEndWindowIndex > MaxWindowIndex THEN
			mEndWindowIndex := mEndWindowIndex - MaxWindowIndex;
		END_IF
		
		mZoneEndPosition := mStartTrackingPosition + mLength;
		
		IF mZoneEndPosition > TotalTrackingLength THEN
			mZoneEndPosition := mZoneEndPosition - TotalTrackingLength;
		END_IF 
		
		ZoneTable[ZoneIndex].Used := TRUE;
		ZoneTable[ZoneIndex].ActionId := mActionId;
		ZoneTable[ZoneIndex].ZoneStartWindowIndex := mStartWindowIndex;
		ZoneTable[ZoneIndex].ZoneStartPosition := mStartTrackingPosition;
		ZoneTable[ZoneIndex].ZoneEndWindowIndex := mEndWindowIndex;
		ZoneTable[ZoneIndex].ZoneEndPosition := mZoneEndPosition;
		ZoneTable[ZoneIndex].ZoneLength := mLength;
		ZoneTable[ZoneIndex].InhibitShifting := mInhibitShifting;
		ZoneTable[ZoneIndex].iActionListener := miActionListener;
		ZoneTable[ZoneIndex].PositionToLive := mPositionToLive;

		IF mPositionToLive > 0 THEN
			M_AddZoneToPTL(ZoneIndex);
		END_IF
		
		// Inform listener
		IF iEventListener <> 0 THEN
			iEventListener.M_TrackingZoneAddedEvent(ZoneIndex,ZoneTable[ZoneIndex]);
		END_IF
		
		M_ReserveZone := ZoneIndex;
	ELSE
		// Error
		fbDebugMsg.M_SendErrorMsg('M_ReserveZone - Could not find free zone.');	
	END_IF
END_IF
END_METHOD

/// This function synchronize only a Front edge to a specific position and calculates the new TU length.
/// Remark: Zone begin gets adjusted to new front edge position. Spare windows in front of front edge get removed.
/// Remark: If at absolute position no zone is found, it searchs to the left for next front edge
/// until "mMaxFrontEdgeDeviation" to synchronize.
METHOD M_ResyncOnlyFE : UINT // Returns > 0 of the synchronized Zone index, otherwise 0 (e.g. No Zone, No occupied zone)
VAR_INPUT
	mAbsolutePosition		: UDINT; // Absolute position [mm]
	mMaxFrontEdgeDeviation 	: UDINT; (* When zone can not be found at "Absolute position",
										a search upwards is executed to a limit of MaxFrontEdgeDeviation [mm]*)
END_VAR
VAR_INST
	MaxTrackingPosition		: UDINT; // Max tracking distance to search for a zone
	NewPositionFE			: UDINT; // New front edge position in tracking
	NumberOfDeviationWindows: UINT; // Number of windows for maximal edge deviation 
	ZoneIndex				: UINT; // Zone index
	ZoneWindowLength 		: UINT; // Length of zone to be moved
	ExistingWindowIndexFE	: UINT; // Existing front edge window index
	ResyncPossible			: BOOL; // Resync is possible
	OldWindowFE				: ST_WindowTrackingWindow; // Stored old front edge window
	DistanceToTU_End		: DINT; // Distance to found TU End
	DistanceToTU_Start		: DINT; // Distance to found TU start
END_VAR
VAR
	mNewWindowIndexFE		: UINT; // Actual window index
	mWindowIndex			: UINT; // Window index iterator
	mIdx					: UINT; // Loop iterator
	mZoneFreeOk				: BOOL; // Shift possible
	mNewZoneWindowLength	: UINT; // Length of windows of aligned zone
END_VAR
M_ResyncOnlyFE := 0;
ZoneIndex := 0;
NumberOfDeviationWindows := 0;
mNewZoneWindowLength := 0;
ResyncPossible := TRUE;

// Validate values
IF WindowSize = 0 THEN
	RETURN;
END_IF

// Get window index at position
mNewWindowIndexFE := M_GetWindowIndex(mAbsolutePosition);

// Find related ZoneIndex
IF mNewWindowIndexFE > 0 AND mNewWindowIndexFE <= WindowTracking.MAX_NUMBER_OF_WINDOWS THEN
	// Ensure that target window is not already a rear edge window 
	// This is not permitted, minimum zone is two window
	IF WindowTable[mNewWindowIndexFE].State = E_WindowTrackingWindowState.REAR_EDGE THEN
		ZoneIndex := 0;
		
